// SIMATIC STEP 7 (V5.x) project AmPackRackWIP
// CPU: CPU 315F-2 PN/DP
// CPU: CPU 315F-2 PN/DP
// CPU: CPU 315F-2 PN/DP
// CPU: CPU 315F-2 PN/DP
// CPU: CPU 315F-2 PN/DP
// CPU: CPU 315F-2 PN/DP
// CPU: CPU 315F-2 PN/DP
// station: P_ADR_BUS
// station: _S7H_BUSSYSTEM_CT
// station: SIMATIC Central
// station: Hardware
// station: P_ADR_BUS
// station: SIMATIC Trolley 1
// station: Hardware
// station: P_ADR_BUS
// station: SIMATIC Carrrier 1
// station: Hardware
// station: P_ADR_BUS
// station: SIMATIC Carrrier 2
// station: Hardware
// station: P_ADR_BUS
// station: SIMATIC Trolley 2
// station: Hardware
// station: P_ADR_BUS
// station: SIMATIC Trolley 3
// station: Hardware
// station: P_ADR_BUS
// station: Konfiguration
// station: Hardware
// station: SIMATIC Pegasus
// station: P_ADR_BUS
// station: _S7H_BUSSYSTEM_CT
// program: S7-TR03
// program: S7-MAIN
// program: S7-TR01
// program: S7-CAR01
// program: S7-CAR02
// program: S7-TR02
// program: S7-Programm(7)

SYMBOL_TABLE
"IDB_SafeMain"	DB 1	FB 1
"DB_BRI"	DB 5	DB 5
"DB_ComGateway"	DB 10	DB 10
"IDB_FB2_BRI"	DB 11	FB 2
"DB_OrderBuffer"	DB 15	DB 15
"DB_TargetData"	DB 19	DB 19
"IDB_MasterInterface"	DB 33	FB 13
"IDB_WREC_BR"	DB 50	SFB 53
"INOUT"	DB 80	DB 80
"Moves"	DB 101	DB 101
"InstanzDB PNIODiag"	DB 126	FB 126
"InstanzDB STATDiag"	DB 127	DB 127
"DB_Steps"	DB 132	DB 132
"COMM_CAR01"	DB 150	DB 150
"BRI_Positions"	DB 200	DB 200
"ProfiNET"	DB 400	DB 400
"Error_Safety"	DB 410	DB 410
"IDB_ESTOP1"	DB 415	FB 215
"F_GLOBDB"	DB 545	DB 545	// F_: F_Global_Data Block
"F00020_4FDI_4FDO_iPar"	DB 546	FB 272
"F00025_4FDI_iPar"	DB 547	FB 272
"DB_GLOBAL"	DB 550	DB 550
"F_IO"	DB 690	DB 690
"F_GBL_RECV"	DB 750	DB 750
"IDB_F_RCV"	DB 751	FB 226
"F_GBL_SEND"	DB 752	DB 752
"IDB_F_SND"	DB 753	FB 225
"IDB_WagoiPar_BRI"	DB 920	FB 37
"DB_iPar_Diag"	DB 930	FB 101
"iPar_Data_Bridge"	DB 1920	DB 1920
"SafeMain"	FB 1	FB 1
"MovidriveB_Control"	FB 2	FB 2
"MasterInterface"	FB 13	FB 13
"CheckEncoder"	FB 21	FB 21
"WAGO_iPar_UDL_4_Mod"	FB 37	FB 37	// WAGO up- / download iParameter PROFIsafe Modules
"TSEND"	FB 63	FB 63	// Send Data
"TRCV"	FB 64	FB 64	// Receive Data
"TCON"	FB 65	FB 65	// Connect
"TDISCON"	FB 66	FB 66	// Disconnect
"Safety_Position"	FB 70	FB 70	// Sichere Positionsüberwachung
"Safety_Direction"	FB 72	FB 72	// Sichere Richtungserfassung
"Safety_Speed"	FB 73	FB 73	// Sichere Geschwindigkeit
"Safety_SpeedCheck"	FB 74	FB 74
"Wago_Bridge"	FB 80	FB 80
"F_Input_MAP"	FB 91	FB 91
"ESTOP"	FB 92	FB 92
"GetPos"	FB 93	FB 93
"DiagPROFIsafe_V2_iPar"	FB 101	FB 101	// read diagnosis data of PROFIsafe modules V2 iPar
"PNIODiag"	FB 126	FB 126	// Profibus/DP und Profinet/IO-Diagnose
"STATDiag"	FB 127	FB 127	// Zweitbaustein (PNIODiag)
"F_TON"	FB 185	FB 185	// F_: Timer Switch On Delay
"F_TOF"	FB 186	FB 186	// F_: Timer Switch Off Delay
"F_ESTOP1"	FB 215	FB 215	// F_: Emergency Stop / Stop Category 1
"F_ACK_GL"	FB 219	FB 219	// F_: Global Acknowledgement of all F-I/O of a RTG
"F_SENDS7"	FB 225	FB 225	// F_: Send S7 Connection
"F_RCVS7"	FB 226	FB 226	// F_: Receive S7 Connection
"F_IO_CGP"	FB 272	FB 272	// F_: Driver Block In-Output with Channel Granular Passivation
"F_CTRL_1"	FB 273	FB 273
"F_CTRL_2"	FB 274	FB 274	// F_: Test Block an Programm Run Control
"F_DIAG_N"	FB 275	FB 275	// F_: Diagnosticbuffer Message with non CPU-Stop
"FITON"	FB 276	FB 276	// FI: Timer Switch On Delay
"FITOF"	FB 277	FB 277	// FI: Timer Switch Off Delay
"FIACK_GL"	FB 278	FB 278	// FI: Global Acknowledgement of all F-I/O of a RTG
"F-CALL"	FC 1	FC 1
"Init"	FC 2	FC 2
"AG_SEND"	FC 5	FC 5	// AG SEND
"AG_RECV"	FC 6	FC 6	// AG RECEIVE
"DT_TOD"	FC 8	FC 8	// DT to TOD
"OpHours"	FC 9	FC 9
"EQ_STRNG"	FC 10	FC 10	// Equal String
"AbsEncoder"	FC 11	FC 11
"DT to DATE"	FC 15	FC 15	// DT to DATE
"Inputs"	FC 30	FC 30
"Outputs"	FC 31	FC 31
"Errors"	FC 40	FC 40
"Errors Reset"	FC 41	FC 41
"Errors_001-016_GEN1"	FC 42	FC 42
"Errors_017-032_GEN2"	FC 43	FC 43
"Errors_033-048_NET"	FC 44	FC 44
"EOff_MachineOff"	FC 48	FC 48
"OP_Mode"	FC 49	FC 49
"Send_Buffer"	FC 52	FC 52
"MSG_161-176"	FC 55	FC 55
"MSG_177_192"	FC 56	FC 56
"CheckWindowDi"	FC 100	FC 100
"Communication"	FC 103	FC 103
"STEPS_Control"	FC 110	FC 110
"STEPS_OrderData"	FC 111	FC 111
"STEPS_EMPTY"	FC 113	FC 113
"Axis_BRIDGE"	FC 200	FC 200
"Axis_BRIDGE_Release"	FC 201	FC 201
"Axis_BRIDGE_Control"	FC 202	FC 202
"Axis_BRIDGE_Speed"	FC 203	FC 203
"Axis_BRIDGE_Scan"	FC 204	FC 204
"Axis_BRIDGE_ScanMan"	FC 205	FC 205
"Axis_BRIDGE_Flt_049-064"	FC 209	FC 209
"iPar_ServerCall"	FC 900	FC 900
"BRIGetPosVal_New"	FC 1071	FC 1071
"I_BRI_EStop"	I 20.0	BOOL	// Emergency-Stop tripped
"I_BRI_FB_FastStop"	I 20.1	BOOL	// Feedback safestop bridge
"I_BRI_FB_EStop_CH1"	I 20.2	BOOL	// Feedback E-Stop  CH1
"I_BRI_FB_EStop_CH2"	I 20.3	BOOL	// Feedback E-Stop CH2
"I_BRI_TROinParkp_CH1"	I 25.0	BOOL	// Trolley in Park position CH1
"I_BRI_TROinParkp_CH2"	I 25.1	BOOL	// Trolley in Park position CH1
"I_BRI_Brake_OK"	I 25.2	BOOL	// Temperature Brake resistors OK
"E      25.3"	I 25.3	BOOL	// spare
"I_BRI_BTN_Preset"	I 65.0	BOOL	// preset button
"I_BRI_Fuse24VOK"	I 65.1	BOOL	// fuse 24V DC OK
"I_BRI_temp_cabinet_high"	I 65.2	BOOL	// high temperature cabinet
"I_BRI_Power_BrakesOK"	I 65.3	BOOL	// Power supply brakes OK
"I_BRI_Power_480_OK"	I 65.4	BOOL	// Power supply 480V OK
"I_BRI_Power_Fan"	I 65.5	BOOL	// Power supply fan OK
"I_BRI_BTN_Reset"	I 65.6	BOOL	// reset button
"I_BRI_Fan_active"	I 65.7	BOOL	// Fan is active
"I_BRI_LimitSw_Plus"	I 66.0	BOOL	// Bridge : Limit-Switch Plus
"I_BRI_LimitSw_Minus"	I 66.1	BOOL	// Bridge : Limit-Switch Minus
"I_BRI_FS_PlusNO"	I 66.2	BOOL	// Bridge : forced speed reduction Plus NO
"I_BRI_FS_PlusNC"	I 66.3	BOOL	// Bridge : forced speed reduction Plus NC
"I_BRI_FS_MinusNO"	I 66.4	BOOL	// Bridge : forced speed reduction Minus NO
"I_BRI_FS_MinusNC"	I 66.5	BOOL	// Bridge : forced speed reduction Minus NC
"E      66.6"	I 66.6	BOOL	// spare
"E      66.7"	I 66.7	BOOL	// spare
"E      67.0"	I 67.0	BOOL	// temp. RC plus
"E      67.1"	I 67.1	BOOL	// temp. RC minus
"E      67.2"	I 67.2	BOOL	// temp. RC fast plus
"E      67.3"	I 67.3	BOOL	// temp. RC fast minus
"E      67.4"	I 67.4	BOOL	// spare
"E      67.5"	I 67.5	BOOL	// spare
"E      67.6"	I 67.6	BOOL	// spare
"E      67.7"	I 67.7	BOOL	// spare
"I_BR_ABS_Encoder"	ID 220	DWORD
"OFF"	M 0.0	BOOL	// immer aus
"ON"	M 0.1	BOOL	// immer ein
"FIRST_RUN"	M 0.7	BOOL
"ModeService"	M 1.0	BOOL
"ModeManual"	M 1.1	BOOL
"ModeAuto"	M 1.2	BOOL
"ModeBypass"	M 1.3	BOOL
"ModeServiceOrManual"	M 1.4	BOOL
"StartAuto"	M 1.5	BOOL
"ModeAutoOrManual"	M 1.6	BOOL
"LifeBitMasterOK"	M 1.7	BOOL
"Eoff"	M 2.0	BOOL
"DivEoff"	M 2.1	BOOL
"Error"	M 2.2	BOOL
"Safty_Vorne"	M 2.4	BOOL
"Safty_Hinten"	M 2.5	BOOL
"Safty_Area"	M 2.6	BOOL
"EmOffRelais_delayed"	M 3.0	BOOL
"Clock0_1"	M 10.0	BOOL	// CPU-Takt 0,1s
"Clock0_2"	M 10.1	BOOL	// CPU-Takt 0,2s
"Clock0_4"	M 10.2	BOOL	// CPU-Takt 0,4s
"Clock0_5"	M 10.3	BOOL	// CPU-Takt 0,5s
"Clock0_8"	M 10.4	BOOL	// CPU-Takt 0,8s
"Clock1_0"	M 10.5	BOOL	// CPU-Takt 1,0s
"Clock1_6"	M 10.6	BOOL	// CPU-Takt 1,6s
"Clock2_0"	M 10.7	BOOL	// CPU-Takt 2,0s
"Tick0_1"	M 11.0	BOOL	// Impuls 0,1s
"Tick0_2"	M 11.1	BOOL	// Impuls 0,2s
"Tick0_4"	M 11.2	BOOL	// Impuls 0,4s
"Tick0_5"	M 11.3	BOOL	// Impuls 0,6s
"Tick0_8"	M 11.4	BOOL	// Impuls 0,8s
"Tick1_0"	M 11.5	BOOL	// Impuls 1,0s
"Tick1_6"	M 11.6	BOOL	// Impuls 1,6s
"Tick2_0"	M 11.7	BOOL	// Impuls 2,0s
"SysPulse_0_1"	M 12.0	BOOL
"SysPulse_0_2"	M 12.1	BOOL
"SysPulse_0_4"	M 12.2	BOOL
"SysPulse_0_5"	M 12.3	BOOL
"SysPulse_0_8"	M 12.4	BOOL
"SysPulse_1_0"	M 12.5	BOOL
"SysPulse_1_6"	M 12.6	BOOL
"SysPulse_2_0"	M 12.7	BOOL
"Next_Step"	M 44.0	BOOL
"SingleStep_ON"	M 44.1	BOOL
"One_Single_Step"	M 44.2	BOOL
"BRI_iPar_Check"	M 920.0	BOOL
"BRI_iPar_UpLoad"	M 920.1	BOOL
"BRI_iPar_DownL"	M 920.2	BOOL
"BRI_iPar_ReqDiag"	M 920.5	BOOL
"pFL_BR_StartWago"	M 925.1	BOOL
"pFL_BR_EndWago"	M 925.2	BOOL
"pFl_ResetErrors"	M 1201.2	BOOL
"pFl_13"	M 1201.3	BOOL
"pFl_14"	M 1201.4	BOOL
"pFl_CNT_StartOrder"	M 1202.0	BOOL
"pFl_CNT_EndOrder"	M 1202.1	BOOL
"pFl_SingleNext"	M 1510.0	BOOL
"Bruno_B"	M 2013.0	BOOL	// Programmpunkt muss noch bearbeitet werden
"bTemp0"	MB 20	BYTE
"diTemp00"	MD 20	DWORD
"ENC_Process"	MD 84	DWORD
"CPY_DATETIME_1"	MD 830	DWORD
"CPY_DATETIME_2"	MD 834	DWORD
"BRI_Pos_Motor"	MD 1000	DWORD
"BRI_Pos_Encoder"	MD 1004	DWORD
"CntMsg"	MW 120	INT
"BRI_Motor_HIGH"	MW 1000	INT
"BRI_Motor_LOW"	MW 1002	INT
"BRI_Encoder_HIGH"	MW 1004	INT
"BRI_Encoder_LOW"	MW 1006	INT
"Bruno_W1"	MW 2014	WORD	// Schmierwort
"Bruno_W2"	MW 2016	WORD	// Schmierwort
"Cycle"	OB 1	OB 1
"CYC_INT5"	OB 35	OB 35	// Cyclic Interrupt 5
"I/O_FLT1"	OB 82	OB 82	// I/O Point Fault 1
"I/O_FLT2"	OB 83	OB 83	// I/O Point Fault 2
"OBNL_FLT"	OB 85	OB 85	// OB Not Loaded Fault
"RACK_FLT"	OB 86	OB 86	// Loss of Rack Fault
"COMM_FLT"	OB 87	OB 87	// Communication Fault
"STARTUP"	OB 100	OB 100
"PROG_ERR"	OB 121	OB 121	// Programming Error
"MOD_ERR"	OB 122	OB 122	// Module Access Error
"A      20.0"	Q 20.0	BOOL	// spare
"O_BRI_SafeStop"	Q 20.1	BOOL	// Fast-Stop bridge
"O_BRI_SafeEStop_CH1"	Q 20.2	BOOL	// E-Stop bridge CH1
"O_BRI_SafeEStop_CH2"	Q 20.3	BOOL	// E-Stop bridge CH2
"O_BRI_LP_Preset"	Q 65.0	BOOL	// lamp preset button
"O_BRI_Reset_24V"	Q 65.1	BOOL	// fuse 24VDC reset
"O_BRI_Reset_EStop"	Q 65.2	BOOL	// EStop reset
"O_BRI_LP_Reset"	Q 65.3	BOOL	// lamp reset button
"O_BRI_Horn"	Q 65.4	BOOL	// startup warning
"O_BRI_State_0"	Q 65.5	BOOL	// lamp state 0
"O_BRI_State_1"	Q 65.6	BOOL	// lamp state 1
"O_BRI_State_2"	Q 65.7	BOOL	// lamp state 2
"TON"	SFB 4	SFB 4	// Generate an On Delay
"USEND"	SFB 8	SFB 8	// Uncoordinated Sending of Data
"URCV"	SFB 9	SFB 9	// Uncoordinated Receiving of Data
"RDREC"	SFB 52	SFB 52	// Read a Process Data Record
"WRREC"	SFB 53	SFB 53	// Write a Process Data Record
"RALRM"	SFB 54	SFB 54	// Receive Alarm Data
"GADR_LGC"	SFC 5	SFC 5	// Query Logical Address of a Channel
"RD_SINFO"	SFC 6	SFC 6	// Read OB Start Information
"D_ACT_DP"	SFC 12	SFC 12	// Deactivating and Activating DP Slaves
"DPNRM_DG"	SFC 13	SFC 13	// Read Diagnostic Data of a DP Slave
"DPRD_DAT"	SFC 14	SFC 14	// Read Consistent Data of a Standard DP Slave
"DPWR_DAT"	SFC 15	SFC 15	// Write Consistent Data to a Standard DP Slave
"BLKMOV"	SFC 20	SFC 20	// Copy Variables
"FILL"	SFC 21	SFC 21	// Initialize a Memory Area
"CREAT_DB"	SFC 22	SFC 22	// Create Data Block
"DEL_DB"	SFC 23	SFC 23	// Delete Data Block
"TEST_DB"	SFC 24	SFC 24	// Test Data Block
"DIS_AIRT"	SFC 41	SFC 41	// Delay the Higher Priority Interrupts and Asynchronous Errors
"EN_AIRT"	SFC 42	SFC 42	// Enable Higher Priority Interrupts and Asynchronous Errors
"STP"	SFC 46	SFC 46	// Change the CPU to STOP
"LGC_GADR"	SFC 49	SFC 49	// Query the Module Slot Belonging to a Logical Address
"RDSYSST"	SFC 51	SFC 51	// Read a System Status List or Partial List
"WR_REC"	SFC 58	SFC 58	// Write Data Record
"RD_REC"	SFC 59	SFC 59	// Read a Data Record
"TIME_TCK"	SFC 64	SFC 64	// Read the System Time
"GEO_LOG"	SFC 70	SFC 70	// Determine Logical Address
"LOG_GEO"	SFC 71	SFC 71	// Determine Geographical Address
"tPlcOn"	T 1	TIMER
"tAknowl"	T 2	TIMER
"t_DelEmOffRelais_1"	T 10	TIMER
"t_DelEmOffRelais_2"	T 11	TIMER
"t_BRIDelFastStop"	T 14	TIMER
"t_BRIDelayInPos"	T 15	TIMER
"t_BRIChkRuntime"	T 16	TIMER
"S_Ev_Mes_Auto"	T 18	TIMER
"T_BRI_Preset_SEW"	T 30	TIMER
"T_Delay:PN_01"	T 40	TIMER
"T_Delay:PN_02"	T 41	TIMER
"T_Delay:PN_03"	T 42	TIMER
"t_DelayReadyOnline"	T 60	TIMER
"t_STEPS_start_DEL"	T 70	TIMER
"T_Startup_Warning"	T 94	TIMER
"T_Startup_Horn"	T 95	TIMER
"T_Check_BRI_FS_Minus"	T 150	TIMER
"T_Check_BRI_FS_Plus"	T 151	TIMER
"t_Err_012"	T 212	TIMER
"t_Err_015"	T 215	TIMER
"t_BRI_EStop"	T 220	TIMER
"OneMove"	UDT 7	UDT 7
"HookData"	UDT 100	UDT 100
"HookDataSheet"	UDT 102	UDT 102
"PosCarrier"	VAT 1	
"TestAuto"	VAT 2	
"TestAGV"	VAT 3	
END_SYMBOL_TABLE

TYPE "OneMove"	// UDT 7
VERSION : 0.1
  STRUCT
   MsgCounter : INT ;
   Action : INT ;
   Value_01 : INT ;
   Value_02 : INT ;
   Value_03 : INT ;
   Value_04 : INT ;
   Value_05 : INT ;
   Value_06 : INT ;
   Value_07 : INT ;
   Value_08 : INT ;
   Value_09 : INT ;
   Value_10 : INT ;
   CRC : INT ;
  END_STRUCT ;	
END_TYPE

TYPE "HookData"	// UDT 100
VERSION : 0.1
  STRUCT
   HookType : INT ;
   TotLengthMin : INT ;
   TotLengthMax : INT ;
   FaceLengthMax : INT ;
   CircumMax : INT ;
   TelPos : DINT ;
   Reserve1 : INT ;
  END_STRUCT ;	
END_TYPE

TYPE "HookDataSheet"	// UDT 102
VERSION : 0.1
  STRUCT
   HookOver : DINT ;
   HookUnderOffset : DINT ;
   TelPos_1 : UDT 100;
   TelPos_2 : UDT 100;
   TelPos_3 : UDT 100;
  END_STRUCT ;	
END_TYPE

FUNCTION_BLOCK "SafeMain"	// FB 1
TITLE = Safe Main
AUTHOR : Koenig
VERSION : 0.1
VAR
  ON : BOOL ;
  M_Reset : BOOL ;
  M_Automatic : BOOL ;
  HardwareOK : BOOL ;
  StateOK : BOOL ;
  ESTOP : BOOL ;
  ESTOP_DEL : BOOL ;
  Release_Bridge : BOOL ;
  BRI_STO : BOOL ;
  BRI_Valid : BOOL ;
  BRI_Work : BOOL ;
  Release_STO : BOOL ;
  nFL_STO : BOOL ;
  BRI_SafeAxis : INT ;
  BRI_Pos : INT ;
  ResetGBL : BOOL ;
  RequestGBL : BOOL ;
  SubsGBL : BOOL ;
  WagoBridge : FB 80;
  F_IO : FB 91;
  E_Stop : FB 92;
  ACK : FB 219;
  TOF_STO : FB 186;
  BRI_SafePos : FB 70;
  T_Reset_GBL : FB 185;
  GetPosCarrier : FB 93;
  ErrorArea : BOOL ;
END_VAR
BEGIN
// body was compiled from another editor; compiled code not shown
END_FUNCTION_BLOCK

FUNCTION_BLOCK "MovidriveB_Control"	// FB 2
TITLE = MovidriveB_Control
//main control for the SEW controller
//KNOW_HOW_PROTECT 
//
AUTHOR : Koenig
VERSION : 0.1
VAR_INPUT
  StateWord : INT ;
  FastStop : BOOL ;
  Reset : BOOL ;
  Start : BOOL ;
  InchMinus : BOOL ;
  InchPlus : BOOL ;
  ModeService : BOOL ;
  ModeAuto : BOOL ;
  ModeRef : BOOL ;
  Bypass : BOOL ;
  PlcOn : BOOL ;
  Pulse_1_0 : BOOL ;
  Tick_0_1 : BOOL ;
  ActualPosition : DINT ;
  TargetPosition : DINT ;
  TargetPositionNo : INT ;
  LimitPlus : DINT ;
  LimitMinus : DINT ;
  InPosWin : DINT ;
END_VAR
VAR_OUTPUT
  CrtWord : INT ;
  Moves : BOOL ;
  Ready : BOOL ;
  RefOk : BOOL ;
  InPos : BOOL ;
  BrakeOpen : BOOL ;
  Error : BOOL ;
  ErrCode : INT ;
  ActPosition : DINT ;
  ActPositionNo : INT ;
  ActTarget : DINT ;
END_VAR
VAR
  INT_iCntRelHalt : INT ;
  INT_iCntInPos : INT ;
  INT_ActualPosition : DINT ;
  INT_ActualPositionNo : INT ;
  INT_pFl_ResetPosition : BOOL ;
  INT_TargetOK : BOOL ;
END_VAR
VAR_TEMP
  INT_xStateCode00 : BOOL ;
  INT_xStateCode01 : BOOL ;
  INT_xStateCode02 : BOOL ;
  INT_xStateCode03 : BOOL ;
  INT_xStateCode04 : BOOL ;
  INT_xStateCode05 : BOOL ;
  INT_xStateCode06 : BOOL ;
  INT_xStateCode07 : BOOL ;
  INT_xState : BOOL ;
  INT_xStateReady : BOOL ;
  INT_xStateRefOk : BOOL ;
  INT_xStateInPos : BOOL ;
  INT_xStateNgrNull : BOOL ;
  INT_xStateErrWarn : BOOL ;
  INT_xStateLimitRight : BOOL ;
  INT_xStateLimitLeft : BOOL ;
  INT_xCrtStart : BOOL ;
  INT_xCrtInchPlus : BOOL ;
  INT_xCrtInchMinus : BOOL ;
  INT_xCrtMode11 : BOOL ;
  INT_xCrtMode12 : BOOL ;
  INT_xCrt13 : BOOL ;
  INT_xCrt14 : BOOL ;
  INT_xCrtBypassLimits : BOOL ;
  INT_xCrtLock : BOOL ;
  INT_xCrtRelFaststop : BOOL ;
  INT_xCrtRelHalt : BOOL ;
  INT_xCrtNotPosCrt : BOOL ;
  INT_xCrtRampsSet2 : BOOL ;
  INT_xCrtParaSet2 : BOOL ;
  INT_xCrtReset : BOOL ;
  INT_xCrt06 : BOOL ;
  INT_xModeMan : BOOL ;
  INT_xModeAuto : BOOL ;
  INT_xModeRef : BOOL ;
  INT_ON : BOOL ;
  INT_w00 : WORD ;
  mValue : DINT ;
  pValue : DINT ;
END_VAR
BEGIN
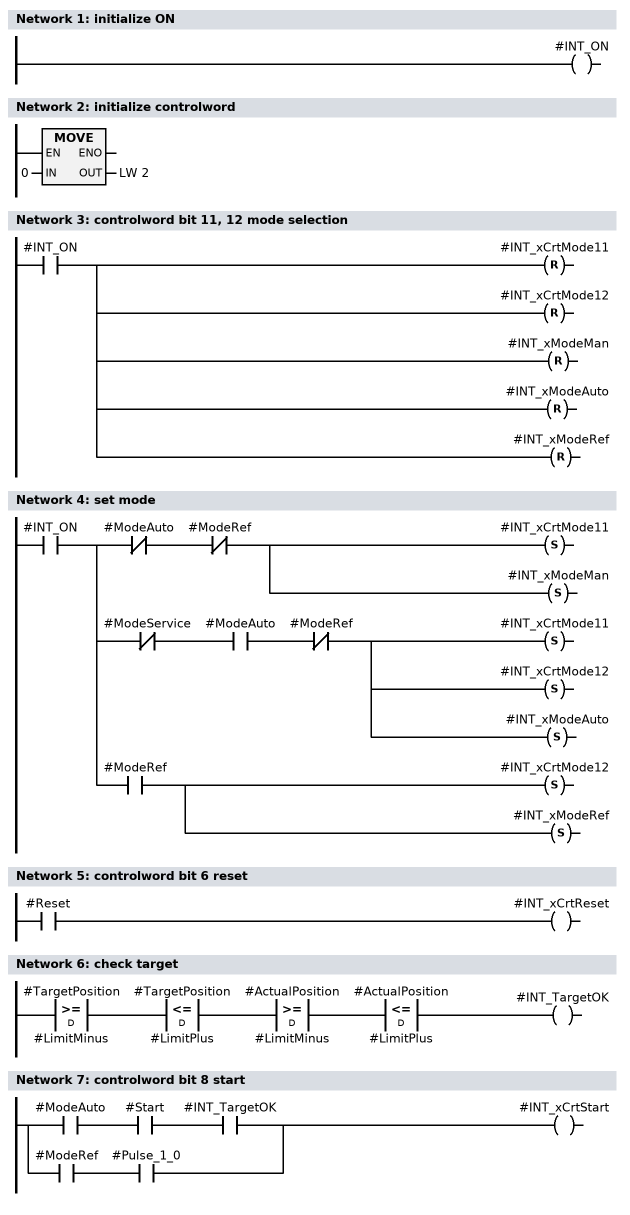
NETWORK
TITLE = initialize ON
//LW0: controler state word
//LW2: controler control word
      SET;
      =     #INT_ON;
NETWORK
TITLE = initialize controlword
      L     0;
      T     LW 2;
      NOP   0;
NETWORK
TITLE = controlword bit 11, 12 mode selection
      A     #INT_ON;
      R     #INT_xCrtMode11;
      R     #INT_xCrtMode12;
      R     #INT_xModeMan;
      R     #INT_xModeAuto;
      R     #INT_xModeRef;
NETWORK
TITLE = set mode
      A     #INT_ON;
      =     L 16.0;
      A     L 16.0;
      AN    #ModeAuto;
      AN    #ModeRef;
      S     #INT_xCrtMode11;
      S     #INT_xModeMan;
      A     L 16.0;
      AN    #ModeService;
      A     #ModeAuto;
      AN    #ModeRef;
      S     #INT_xCrtMode11;
      S     #INT_xCrtMode12;
      S     #INT_xModeAuto;
      A     L 16.0;
      A     #ModeRef;
      S     #INT_xCrtMode12;
      S     #INT_xModeRef;
NETWORK
TITLE = controlword bit 6 reset
      A     #Reset;
      =     #INT_xCrtReset;
NETWORK
TITLE = check target
      A(;
      L     #TargetPosition;
      L     #LimitMinus;
      >=D;
      );
      A(;
      L     #TargetPosition;
      L     #LimitPlus;
      <=D;
      );
      A(;
      L     #ActualPosition;
      L     #LimitMinus;
      >=D;
      );
      A(;
      L     #ActualPosition;
      L     #LimitPlus;
      <=D;
      );
      =     #INT_TargetOK;
NETWORK
TITLE = controlword bit 8 start
      A     #ModeAuto;
      A     #Start;
      A     #INT_TargetOK;
      O;
      A     #ModeRef;
      A     #Pulse_1_0;
      =     #INT_xCrtStart;
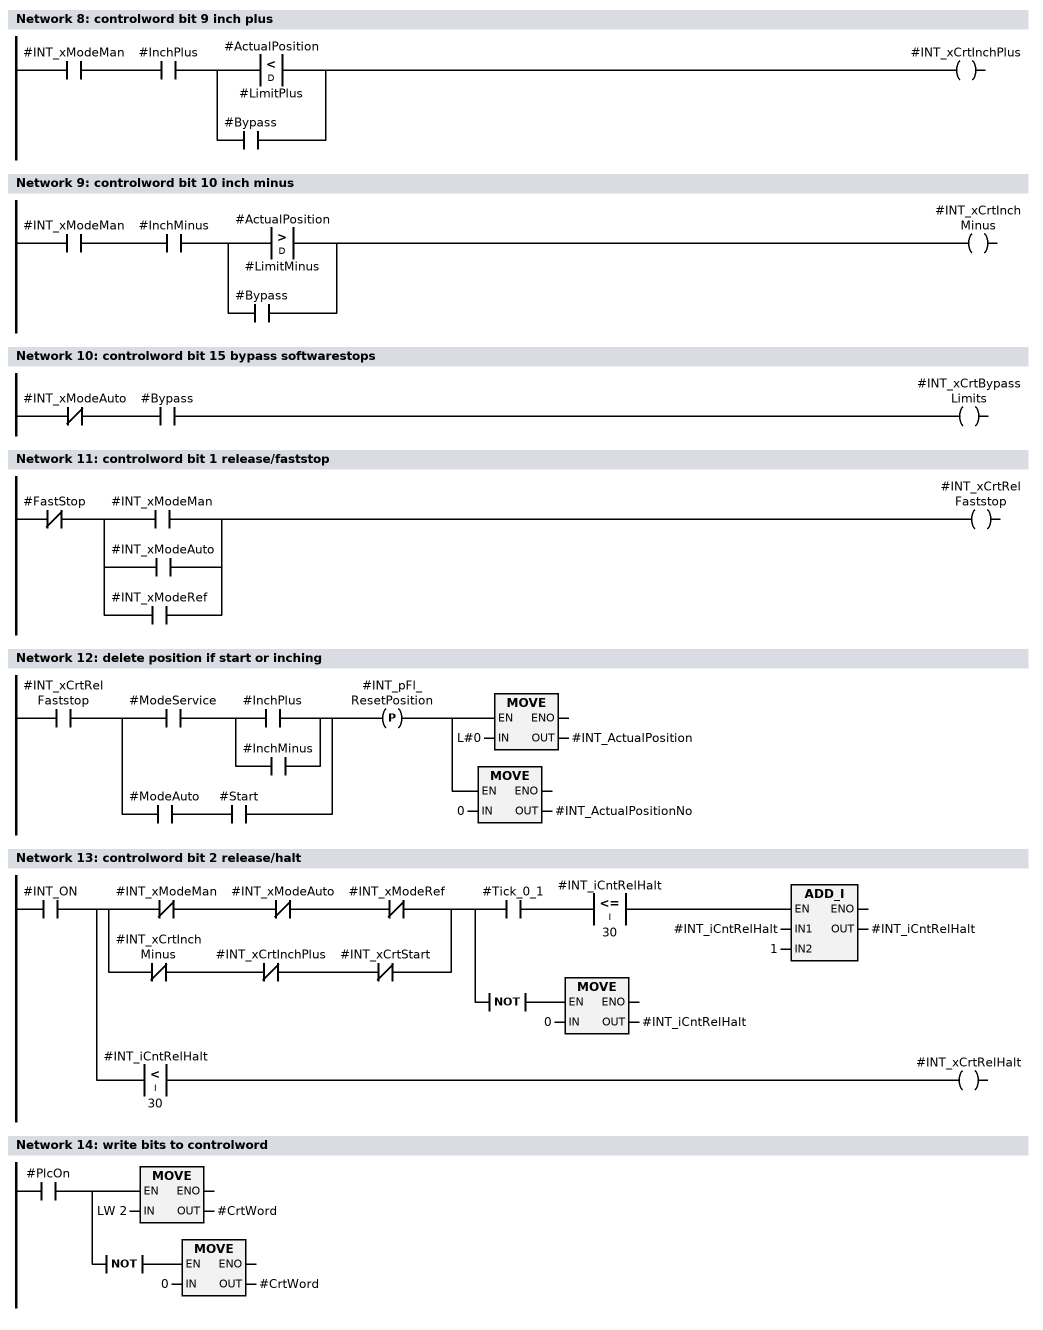
NETWORK
TITLE = controlword bit 9 inch plus
      A     #INT_xModeMan;
      A     #InchPlus;
      A(;
      O(;
      L     #ActualPosition;
      L     #LimitPlus;
      <D;
      );
      O     #Bypass;
      );
      =     #INT_xCrtInchPlus;
NETWORK
TITLE = controlword bit 10 inch minus
      A     #INT_xModeMan;
      A     #InchMinus;
      A(;
      O(;
      L     #ActualPosition;
      L     #LimitMinus;
      >D;
      );
      O     #Bypass;
      );
      =     #INT_xCrtInchMinus;
NETWORK
TITLE = controlword bit 15 bypass softwarestops
      AN    #INT_xModeAuto;
      A     #Bypass;
      =     #INT_xCrtBypassLimits;
NETWORK
TITLE = controlword bit 1 release/faststop
      AN    #FastStop;
      A(;
      O     #INT_xModeMan;
      O     #INT_xModeAuto;
      O     #INT_xModeRef;
      );
      =     #INT_xCrtRelFaststop;
NETWORK
TITLE = delete position if start or inching
      A     #INT_xCrtRelFaststop;
      A(;
      A     #ModeService;
      A(;
      O     #InchPlus;
      O     #InchMinus;
      );
      O;
      A     #ModeAuto;
      A     #Start;
      );
      FP    #INT_pFl_ResetPosition;
      =     L 16.0;
      A     L 16.0;
      JNB   _001;
      L     L#0;
      T     #INT_ActualPosition;
_001: NOP   0;
      A     L 16.0;
      JNB   _002;
      L     0;
      T     #INT_ActualPositionNo;
_002: NOP   0;
NETWORK
TITLE = controlword bit 2 release/halt
      A     #INT_ON;
      =     L 16.0;
      A     L 16.0;
      A(;
      AN    #INT_xModeMan;
      AN    #INT_xModeAuto;
      AN    #INT_xModeRef;
      O;
      AN    #INT_xCrtInchMinus;
      AN    #INT_xCrtInchPlus;
      AN    #INT_xCrtStart;
      );
      =     L 16.1;
      A     L 16.1;
      A     #Tick_0_1;
      A(;
      L     #INT_iCntRelHalt;
      L     30;
      <=I;
      );
      JNB   _003;
      L     #INT_iCntRelHalt;
      L     1;
      +I;
      T     #INT_iCntRelHalt;
_003: NOP   0;
      A     L 16.1;
      NOT;
      JNB   _004;
      L     0;
      T     #INT_iCntRelHalt;
_004: NOP   0;
      A     L 16.0;
      A(;
      L     #INT_iCntRelHalt;
      L     30;
      <I;
      );
      =     #INT_xCrtRelHalt;
NETWORK
TITLE = write bits to controlword
      A     #PlcOn;
      =     L 16.0;
      A     L 16.0;
      JNB   _005;
      L     LW 2;
      T     #CrtWord;
_005: NOP   0;
      A     L 16.0;
      NOT;
      JNB   _006;
      L     0;
      T     #CrtWord;
_006: NOP   0;
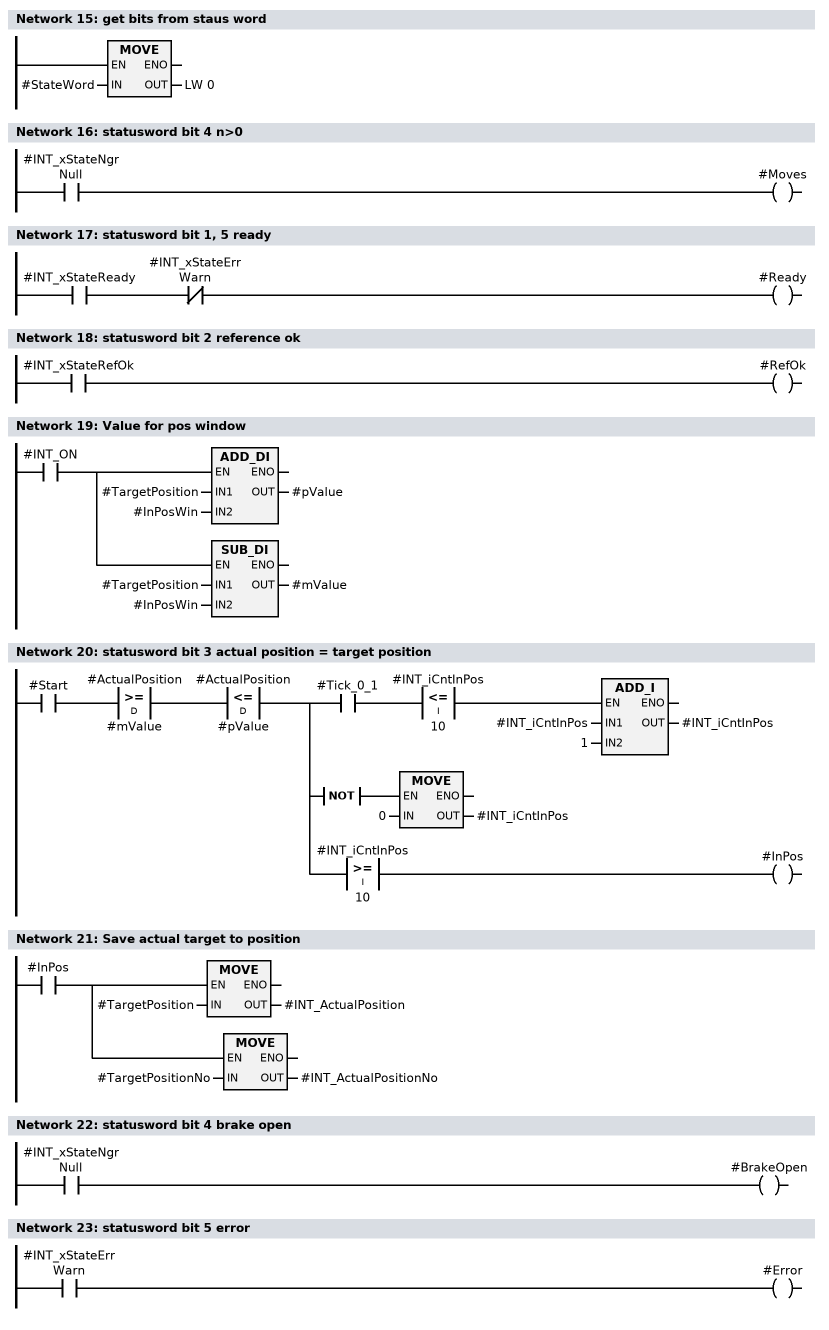
NETWORK
TITLE = get bits from staus word
      L     #StateWord;
      T     LW 0;
      NOP   0;
NETWORK
TITLE = statusword bit 4 n>0
      A     #INT_xStateNgrNull;
      =     #Moves;
NETWORK
TITLE = statusword bit 1, 5 ready
      A     #INT_xStateReady;
      AN    #INT_xStateErrWarn;
      =     #Ready;
NETWORK
TITLE = statusword bit 2 reference ok
      A     #INT_xStateRefOk;
      =     #RefOk;
NETWORK
TITLE = Value for pos window
      A     #INT_ON;
      =     L 16.0;
      A     L 16.0;
      JNB   _007;
      L     #TargetPosition;
      L     #InPosWin;
      +D;
      T     #pValue;
_007: NOP   0;
      A     L 16.0;
      JNB   _008;
      L     #TargetPosition;
      L     #InPosWin;
      -D;
      T     #mValue;
_008: NOP   0;
NETWORK
TITLE = statusword bit 3 actual position = target position
//note: in omron we use the actual position and the target postion equal
//
      A     #Start;
      A(;
      L     #ActualPosition;
      L     #mValue;
      >=D;
      );
      A(;
      L     #ActualPosition;
      L     #pValue;
      <=D;
      );
      =     L 16.0;
      A     L 16.0;
      A     #Tick_0_1;
      A(;
      L     #INT_iCntInPos;
      L     10;
      <=I;
      );
      JNB   _009;
      L     #INT_iCntInPos;
      L     1;
      +I;
      T     #INT_iCntInPos;
_009: NOP   0;
      A     L 16.0;
      NOT;
      JNB   _00a;
      L     0;
      T     #INT_iCntInPos;
_00a: NOP   0;
      A     L 16.0;
      A(;
      L     #INT_iCntInPos;
      L     10;
      >=I;
      );
      =     #InPos;
NETWORK
TITLE = Save actual target to position
      A     #InPos;
      =     L 16.0;
      A     L 16.0;
      JNB   _00b;
      L     #TargetPosition;
      T     #INT_ActualPosition;
_00b: NOP   0;
      A     L 16.0;
      JNB   _00c;
      L     #TargetPositionNo;
      T     #INT_ActualPositionNo;
_00c: NOP   0;
NETWORK
TITLE = statusword bit 4 brake open
      A     #INT_xStateNgrNull;
      =     #BrakeOpen;
NETWORK
TITLE = statusword bit 5 error
      A     #INT_xStateErrWarn;
      =     #Error;
NETWORK
TITLE = status / error code
      A     #INT_ON;
      =     L 16.0;
      A     L 16.0;
      JNB   _00d;
      L     LW 0;
      L     W#16#FF00;
      AW;
      T     LW 0;
_00d: NOP   0;
      A     L 16.0;
      JNB   _00e;
      L     W#16#8;
      L     LW 0;
      SRW;
      T     LW 0;
_00e: NOP   0;
      A     L 16.0;
      JNB   _00f;
      L     LW 0;
      T     #ErrCode;
_00f: NOP   0;
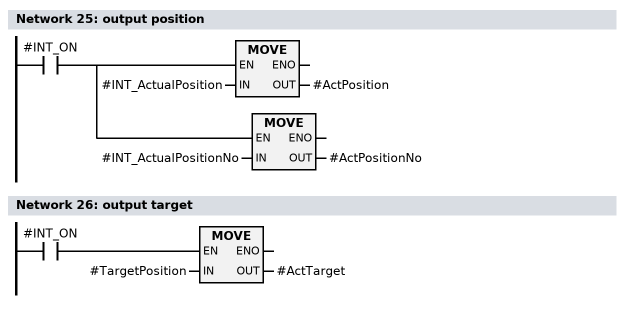
NETWORK
TITLE = output position
      A     #INT_ON;
      =     L 16.0;
      A     L 16.0;
      JNB   _010;
      L     #INT_ActualPosition;
      T     #ActPosition;
_010: NOP   0;
      A     L 16.0;
      JNB   _011;
      L     #INT_ActualPositionNo;
      T     #ActPositionNo;
_011: NOP   0;
NETWORK
TITLE = output target
      A     #INT_ON;
      JNB   _012;
      L     #TargetPosition;
      T     #ActTarget;
_012: NOP   0;
END_FUNCTION_BLOCK

FUNCTION_BLOCK "MasterInterface"	// FB 13
//LW0: control word from master
//LW2: status word to master
VERSION : 0.1
VAR_INPUT
  IN_iCrtWord : INT ;
  IN_iCommCounter : INT ;
  IN_iToggleTime_0_1sec : INT ;
  IN_xFree : BOOL ;
  IN_xOccupied : BOOL ;
  IN_xLiftTop : BOOL ;
  IN_xOnline : BOOL ;
  IN_xReadyOnline : BOOL ;
  IN_xError : BOOL ;
  IN_xMovingSource : BOOL ;
  IN_xMovingTarget : BOOL ;
  IN_x09 : BOOL ;
  IN_xOrderRunning : BOOL ;
  IN_xOrderEnd : BOOL ;
  IN_xOrderPaused : BOOL ;
  IN_x13 : BOOL ;
  IN_xNewTarget : BOOL ;
  IN_x15 : BOOL ;
  IN_SysTick : BOOL ;
END_VAR
VAR_OUTPUT
  OUT_iStateWord : INT ;
  OUT_xLifeBitOk : BOOL ;
  OUT_x01 : BOOL ;
  OUT_xStartBasePos : BOOL ;
  OUT_xStartNewTarget : BOOL ;
  OUT_xAknOrderEnd : BOOL ;
  OUT_xReset : BOOL ;
  OUT_x06 : BOOL ;
  OUT_x07 : BOOL ;
  OUT_x08 : BOOL ;
  OUT_x09 : BOOL ;
  OUT_xStartOrder : BOOL ;
  OUT_xClearOrder : BOOL ;
  OUT_xPauseOrder : BOOL ;
  OUT_x13 : BOOL ;
  OUT_xStartStopPos : BOOL ;
  OUT_xReleaseOnline : BOOL ;
END_VAR
VAR
  INT_b_1 : BOOL ;
  INT_b_2 : BOOL ;
  INT_b_3 : BOOL ;
  INT_iCntLbOn : INT ;
  INT_iCntLbOff : INT ;
  INT_iCntLbOk : INT ;
  INT_iCntStartBasePos : INT ;
  INT_iCntStartNewtarget : INT ;
  INT_iCntStartOrder : INT ;
  INT_iCntStartStopPos : INT ;
  INT_iLastCommCounter : INT ;
  INT_T1 : SFB 4;
  INT_T2 : SFB 4;
END_VAR
VAR_TEMP
  INT_xCrt08 : BOOL ;
  INT_xCrt09 : BOOL ;
  INT_xCrtStartOrder : BOOL ;
  INT_xCrtClearOrder : BOOL ;
  INT_xCrtPauseOrder : BOOL ;
  INT_xCrt13 : BOOL ;
  INT_xCrtStartStopPos : BOOL ;
  INT_xReleaseOnline : BOOL ;
  INT_xCrtLife : BOOL ;
  INT_xCrt01 : BOOL ;
  INT_xCrtStartBasePos : BOOL ;
  INT_xCrtStartNewTarg : BOOL ;
  INT_xCrtAcknOrderEnd : BOOL ;
  INT_xCrtReset : BOOL ;
  INT_xCrt06 : BOOL ;
  INT_xCrt07 : BOOL ;
  INT_xStateMovingTarget : BOOL ;
  INT_xState09 : BOOL ;
  INT_xStateOrderRunning : BOOL ;
  INT_xStateOrderEnd : BOOL ;
  INT_xStateOrderPaused : BOOL ;
  INT_xState13 : BOOL ;
  INT_xStateNewTarget : BOOL ;
  INT_xState15 : BOOL ;
  INT_xStateLife : BOOL ;
  INT_xStateFree : BOOL ;
  INT_xStateOccupied : BOOL ;
  INT_xStateLiftTop : BOOL ;
  INT_xStateOnline : BOOL ;
  INT_xStateReadyOnline : BOOL ;
  INT_xStateError : BOOL ;
  INT_xStateMovingSource : BOOL ;
  ON : BOOL ;
END_VAR
BEGIN
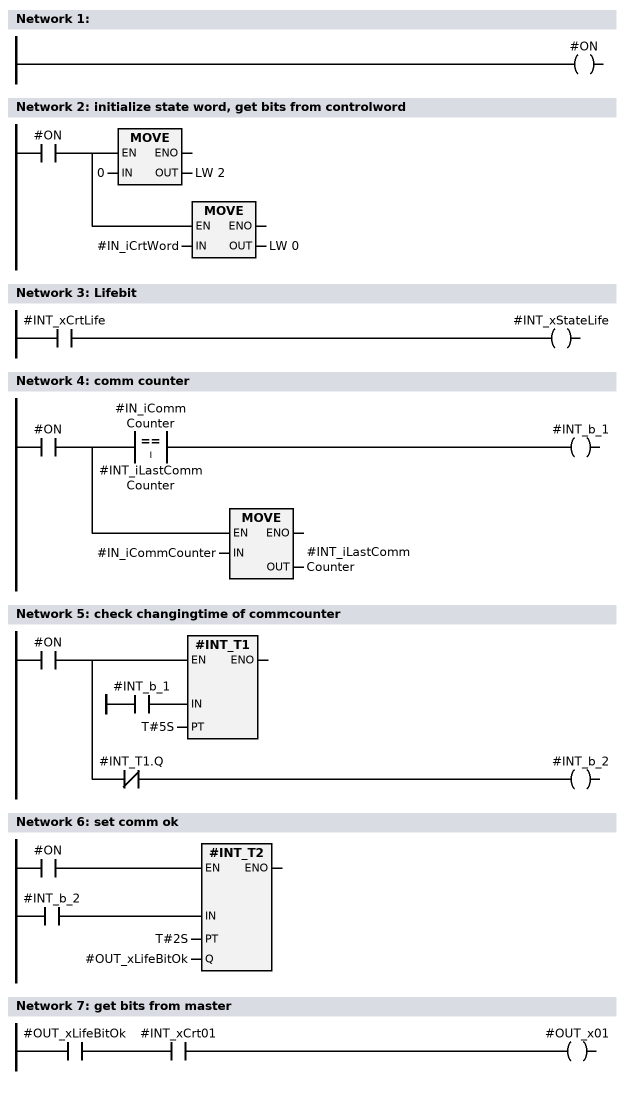
NETWORK
TITLE =
      SET;
      =     #ON;
NETWORK
TITLE = initialize state word, get bits from controlword
      A     #ON;
      =     L 5.0;
      A     L 5.0;
      JNB   _001;
      L     0;
      T     LW 2;
_001: NOP   0;
      A     L 5.0;
      JNB   _002;
      L     #IN_iCrtWord;
      T     LW 0;
_002: NOP   0;
NETWORK
TITLE = Lifebit
      A     #INT_xCrtLife;
      =     #INT_xStateLife;
NETWORK
TITLE = comm counter
      A     #ON;
      =     L 5.0;
      A     L 5.0;
      A(;
      L     #IN_iCommCounter;
      L     #INT_iLastCommCounter;
      ==I;
      );
      =     #INT_b_1;
      A     L 5.0;
      JNB   _003;
      L     #IN_iCommCounter;
      T     #INT_iLastCommCounter;
_003: NOP   0;
NETWORK
TITLE = check changingtime of commcounter
      A     #ON;
      =     L 5.0;
      A     #INT_b_1;
      =     L 5.1;
      BLD   103;
      A     L 5.0;
      JNB   _004;
      CALL  #INT_T1 (
           IN                       := L 5.1,
           PT                       := T#5S);
_004: NOP   0;
      A     L 5.0;
      AN    #INT_T1.Q;
      =     #INT_b_2;
NETWORK
TITLE = set comm ok
      A     #INT_b_2;
      =     L 5.0;
      BLD   103;
      A     #ON;
      JNB   _005;
      CALL  #INT_T2 (
           IN                       := L 5.0,
           PT                       := T#2S,
           Q                        := #OUT_xLifeBitOk);
_005: NOP   0;
NETWORK
TITLE = get bits from master
      A     #OUT_xLifeBitOk;
      A     #INT_xCrt01;
      =     #OUT_x01;
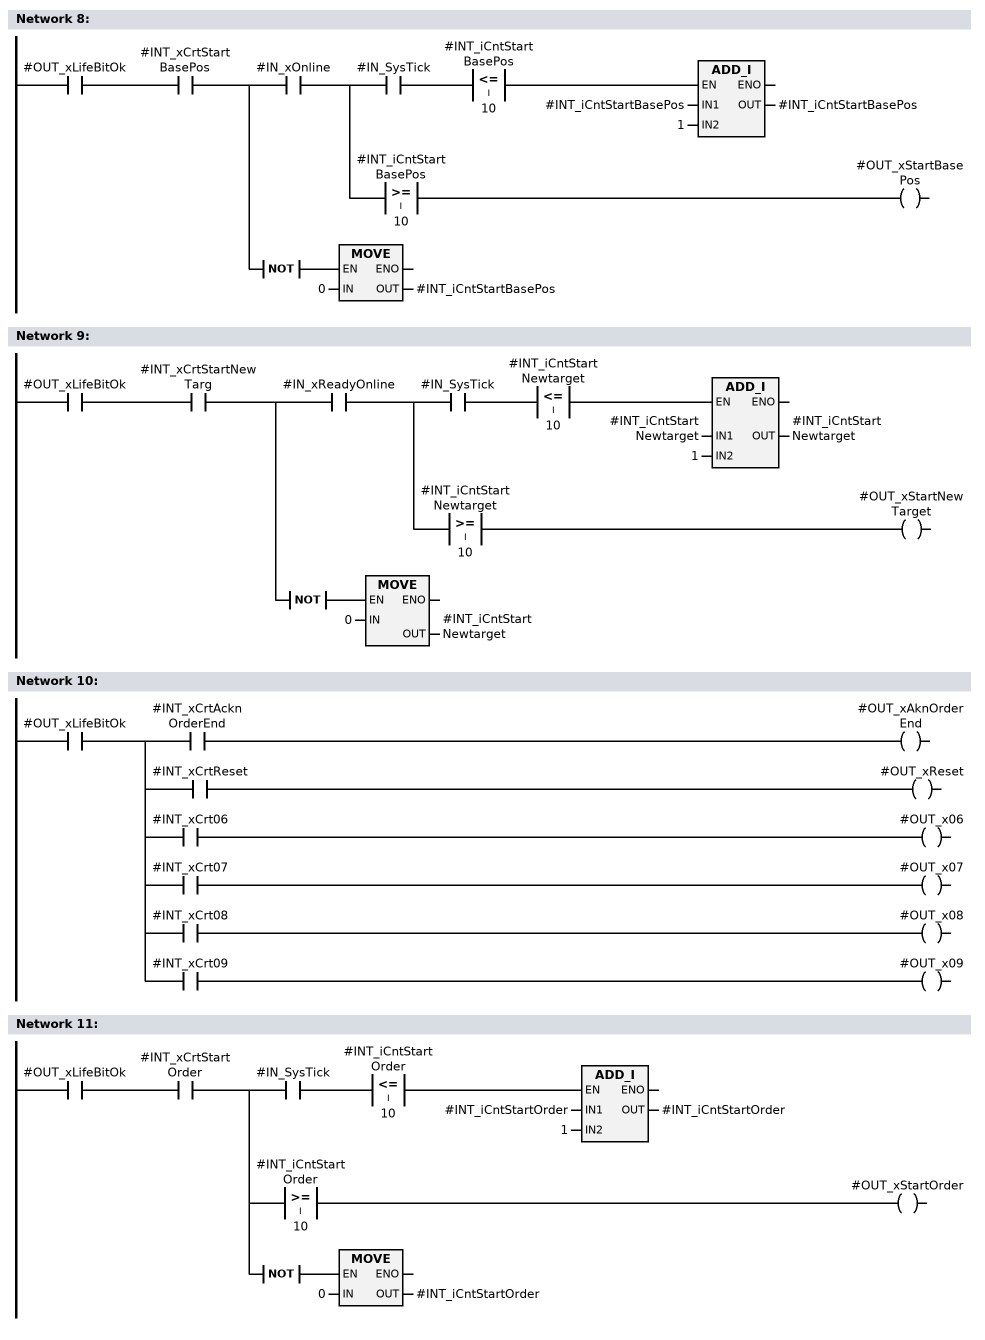
NETWORK
TITLE =
      A     #OUT_xLifeBitOk;
      A     #INT_xCrtStartBasePos;
      =     L 5.0;
      A     L 5.0;
      A     #IN_xOnline;
      =     L 5.1;
      A     L 5.1;
      A     #IN_SysTick;
      A(;
      L     #INT_iCntStartBasePos;
      L     10;
      <=I;
      );
      JNB   _006;
      L     #INT_iCntStartBasePos;
      L     1;
      +I;
      T     #INT_iCntStartBasePos;
_006: NOP   0;
      A     L 5.1;
      A(;
      L     #INT_iCntStartBasePos;
      L     10;
      >=I;
      );
      =     #OUT_xStartBasePos;
      A     L 5.0;
      NOT;
      JNB   _007;
      L     0;
      T     #INT_iCntStartBasePos;
_007: NOP   0;
NETWORK
TITLE =
      A     #OUT_xLifeBitOk;
      A     #INT_xCrtStartNewTarg;
      =     L 5.0;
      A     L 5.0;
      A     #IN_xReadyOnline;
      =     L 5.1;
      A     L 5.1;
      A     #IN_SysTick;
      A(;
      L     #INT_iCntStartNewtarget;
      L     10;
      <=I;
      );
      JNB   _008;
      L     #INT_iCntStartNewtarget;
      L     1;
      +I;
      T     #INT_iCntStartNewtarget;
_008: NOP   0;
      A     L 5.1;
      A(;
      L     #INT_iCntStartNewtarget;
      L     10;
      >=I;
      );
      =     #OUT_xStartNewTarget;
      A     L 5.0;
      NOT;
      JNB   _009;
      L     0;
      T     #INT_iCntStartNewtarget;
_009: NOP   0;
NETWORK
TITLE =
      A     #OUT_xLifeBitOk;
      =     L 5.0;
      A     L 5.0;
      A     #INT_xCrtAcknOrderEnd;
      =     #OUT_xAknOrderEnd;
      A     L 5.0;
      A     #INT_xCrtReset;
      =     #OUT_xReset;
      A     L 5.0;
      A     #INT_xCrt06;
      =     #OUT_x06;
      A     L 5.0;
      A     #INT_xCrt07;
      =     #OUT_x07;
      A     L 5.0;
      A     #INT_xCrt08;
      =     #OUT_x08;
      A     L 5.0;
      A     #INT_xCrt09;
      =     #OUT_x09;
NETWORK
TITLE =
      A     #OUT_xLifeBitOk;
      A     #INT_xCrtStartOrder;
      =     L 5.0;
      A     L 5.0;
      A     #IN_SysTick;
      A(;
      L     #INT_iCntStartOrder;
      L     10;
      <=I;
      );
      JNB   _00a;
      L     #INT_iCntStartOrder;
      L     1;
      +I;
      T     #INT_iCntStartOrder;
_00a: NOP   0;
      A     L 5.0;
      A(;
      L     #INT_iCntStartOrder;
      L     10;
      >=I;
      );
      =     #OUT_xStartOrder;
      A     L 5.0;
      NOT;
      JNB   _00b;
      L     0;
      T     #INT_iCntStartOrder;
_00b: NOP   0;
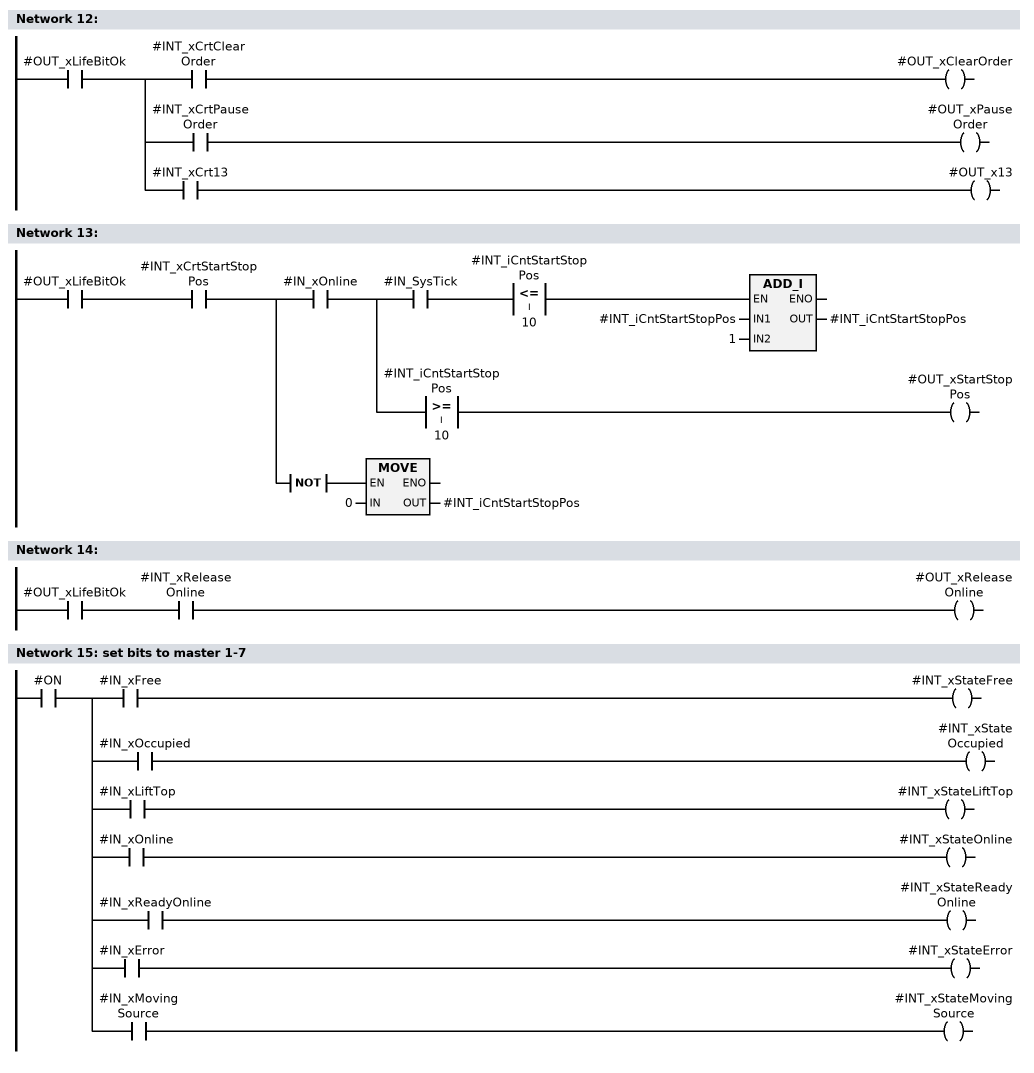
NETWORK
TITLE =
      A     #OUT_xLifeBitOk;
      =     L 5.0;
      A     L 5.0;
      A     #INT_xCrtClearOrder;
      =     #OUT_xClearOrder;
      A     L 5.0;
      A     #INT_xCrtPauseOrder;
      =     #OUT_xPauseOrder;
      A     L 5.0;
      A     #INT_xCrt13;
      =     #OUT_x13;
NETWORK
TITLE =
      A     #OUT_xLifeBitOk;
      A     #INT_xCrtStartStopPos;
      =     L 5.0;
      A     L 5.0;
      A     #IN_xOnline;
      =     L 5.1;
      A     L 5.1;
      A     #IN_SysTick;
      A(;
      L     #INT_iCntStartStopPos;
      L     10;
      <=I;
      );
      JNB   _00c;
      L     #INT_iCntStartStopPos;
      L     1;
      +I;
      T     #INT_iCntStartStopPos;
_00c: NOP   0;
      A     L 5.1;
      A(;
      L     #INT_iCntStartStopPos;
      L     10;
      >=I;
      );
      =     #OUT_xStartStopPos;
      A     L 5.0;
      NOT;
      JNB   _00d;
      L     0;
      T     #INT_iCntStartStopPos;
_00d: NOP   0;
NETWORK
TITLE =
      A     #OUT_xLifeBitOk;
      A     #INT_xReleaseOnline;
      =     #OUT_xReleaseOnline;
NETWORK
TITLE = set bits to master 1-7
      A     #ON;
      =     L 5.0;
      A     L 5.0;
      A     #IN_xFree;
      =     #INT_xStateFree;
      A     L 5.0;
      A     #IN_xOccupied;
      =     #INT_xStateOccupied;
      A     L 5.0;
      A     #IN_xLiftTop;
      =     #INT_xStateLiftTop;
      A     L 5.0;
      A     #IN_xOnline;
      =     #INT_xStateOnline;
      A     L 5.0;
      A     #IN_xReadyOnline;
      =     #INT_xStateReadyOnline;
      A     L 5.0;
      A     #IN_xError;
      =     #INT_xStateError;
      A     L 5.0;
      A     #IN_xMovingSource;
      =     #INT_xStateMovingSource;
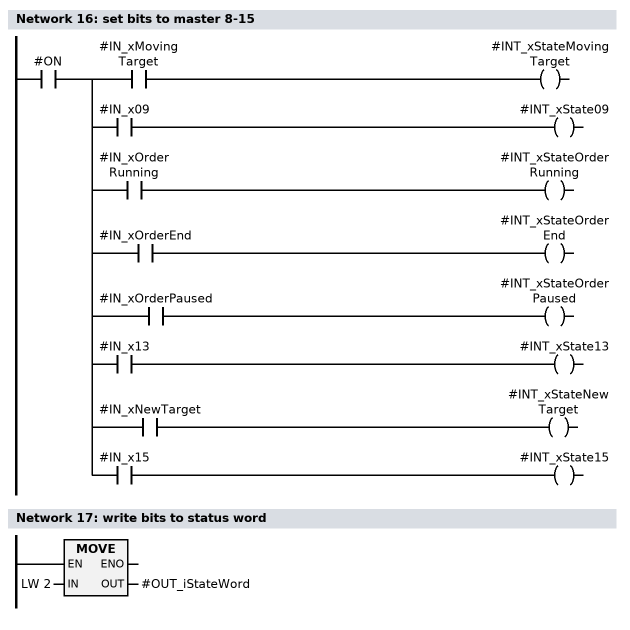
NETWORK
TITLE = set bits to master 8-15
      A     #ON;
      =     L 5.0;
      A     L 5.0;
      A     #IN_xMovingTarget;
      =     #INT_xStateMovingTarget;
      A     L 5.0;
      A     #IN_x09;
      =     #INT_xState09;
      A     L 5.0;
      A     #IN_xOrderRunning;
      =     #INT_xStateOrderRunning;
      A     L 5.0;
      A     #IN_xOrderEnd;
      =     #INT_xStateOrderEnd;
      A     L 5.0;
      A     #IN_xOrderPaused;
      =     #INT_xStateOrderPaused;
      A     L 5.0;
      A     #IN_x13;
      =     #INT_xState13;
      A     L 5.0;
      A     #IN_xNewTarget;
      =     #INT_xStateNewTarget;
      A     L 5.0;
      A     #IN_x15;
      =     #INT_xState15;
NETWORK
TITLE = write bits to status word
      L     LW 2;
      T     #OUT_iStateWord;
      NOP   0;
END_FUNCTION_BLOCK

FUNCTION_BLOCK "CheckEncoder"	// FB 21
TITLE = Check Encoder
VERSION : 0.1
VAR_INPUT
  ActualValue : DINT ;
  TurnMinus : BOOL ;
  TurnPlus : BOOL ;
  Reset : BOOL ;
  Clock_100ms : BOOL ;
  Clock_1s : BOOL ;
  minTurn : DINT ;
  maxTurn : DINT ;
  maxNotTurn : DINT ;
  fadeOut100ms : INT ;
END_VAR
VAR_OUTPUT
  Error : BOOL ;
  ErrorCode : INT ;
END_VAR
VAR
  lastValue : DINT ;
  actDiff : DINT ;
  p_Reset : BOOL ;
  p_Clock : BOOL ;
  p_Clock_1s : BOOL ;
  m_Error : BOOL ;
  timerTurn : INT ;
  timerNotTurn : INT ;
  m_ErrorCode : INT ;
  m_ErrorDiff : DINT ;
  timerCheck : INT ;
END_VAR
VAR_TEMP
  Clock : BOOL ;
  Turn : BOOL ;
  notTurn : BOOL ;
  Clock_1 : BOOL ;
END_VAR
BEGIN
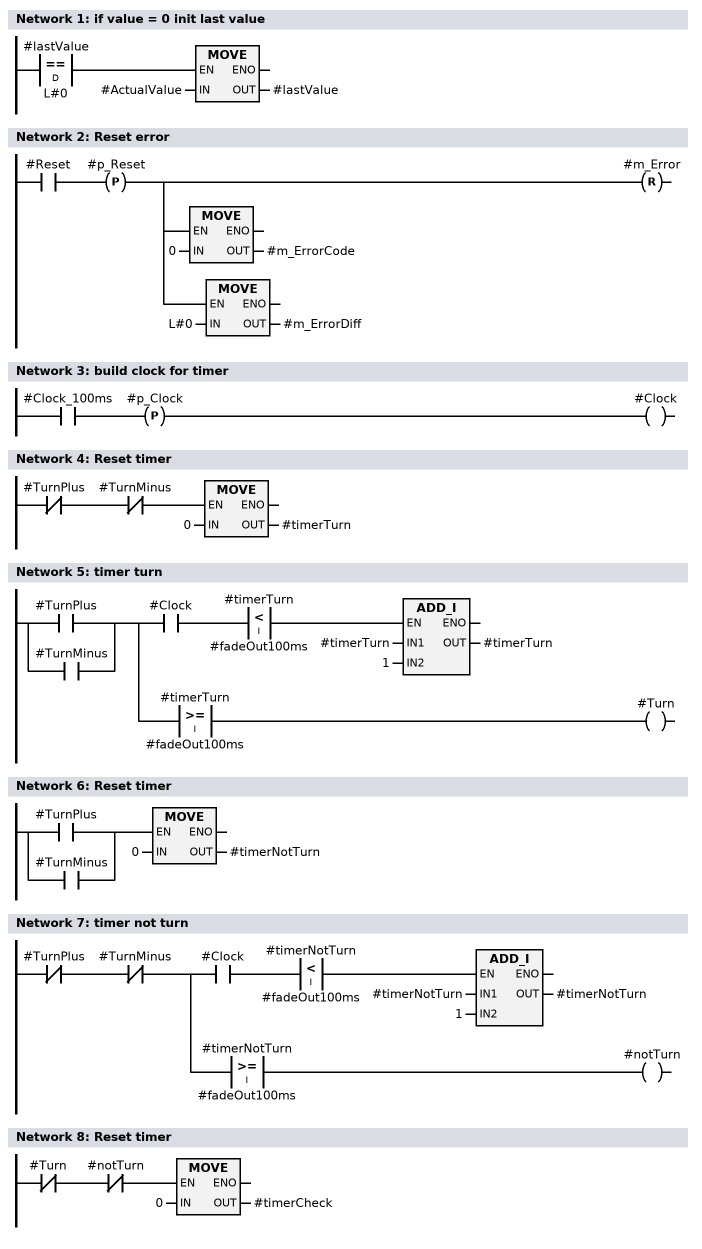
NETWORK
TITLE = if value = 0 init last value
      A(;
      L     #lastValue;
      L     L#0;
      ==D;
      );
      JNB   _001;
      L     #ActualValue;
      T     #lastValue;
_001: NOP   0;
NETWORK
TITLE = Reset error
      A     #Reset;
      FP    #p_Reset;
      =     L 1.0;
      A     L 1.0;
      BLD   102;
      R     #m_Error;
      A     L 1.0;
      JNB   _002;
      L     0;
      T     #m_ErrorCode;
_002: NOP   0;
      A     L 1.0;
      JNB   _003;
      L     L#0;
      T     #m_ErrorDiff;
_003: NOP   0;
NETWORK
TITLE = build clock for timer
      A     #Clock_100ms;
      FP    #p_Clock;
      =     #Clock;
NETWORK
TITLE = Reset timer
      AN    #TurnPlus;
      AN    #TurnMinus;
      JNB   _004;
      L     0;
      T     #timerTurn;
_004: NOP   0;
NETWORK
TITLE = timer turn
      O     #TurnPlus;
      O     #TurnMinus;
      =     L 1.0;
      A     L 1.0;
      A     #Clock;
      A(;
      L     #timerTurn;
      L     #fadeOut100ms;
      <I;
      );
      JNB   _005;
      L     #timerTurn;
      L     1;
      +I;
      T     #timerTurn;
_005: NOP   0;
      A     L 1.0;
      A(;
      L     #timerTurn;
      L     #fadeOut100ms;
      >=I;
      );
      =     #Turn;
NETWORK
TITLE = Reset timer
      A(;
      O     #TurnPlus;
      O     #TurnMinus;
      );
      JNB   _006;
      L     0;
      T     #timerNotTurn;
_006: NOP   0;
NETWORK
TITLE = timer not turn
      AN    #TurnPlus;
      AN    #TurnMinus;
      =     L 1.0;
      A     L 1.0;
      A     #Clock;
      A(;
      L     #timerNotTurn;
      L     #fadeOut100ms;
      <I;
      );
      JNB   _007;
      L     #timerNotTurn;
      L     1;
      +I;
      T     #timerNotTurn;
_007: NOP   0;
      A     L 1.0;
      A(;
      L     #timerNotTurn;
      L     #fadeOut100ms;
      >=I;
      );
      =     #notTurn;
NETWORK
TITLE = Reset timer
      AN    #Turn;
      AN    #notTurn;
      JNB   _008;
      L     0;
      T     #timerCheck;
_008: NOP   0;
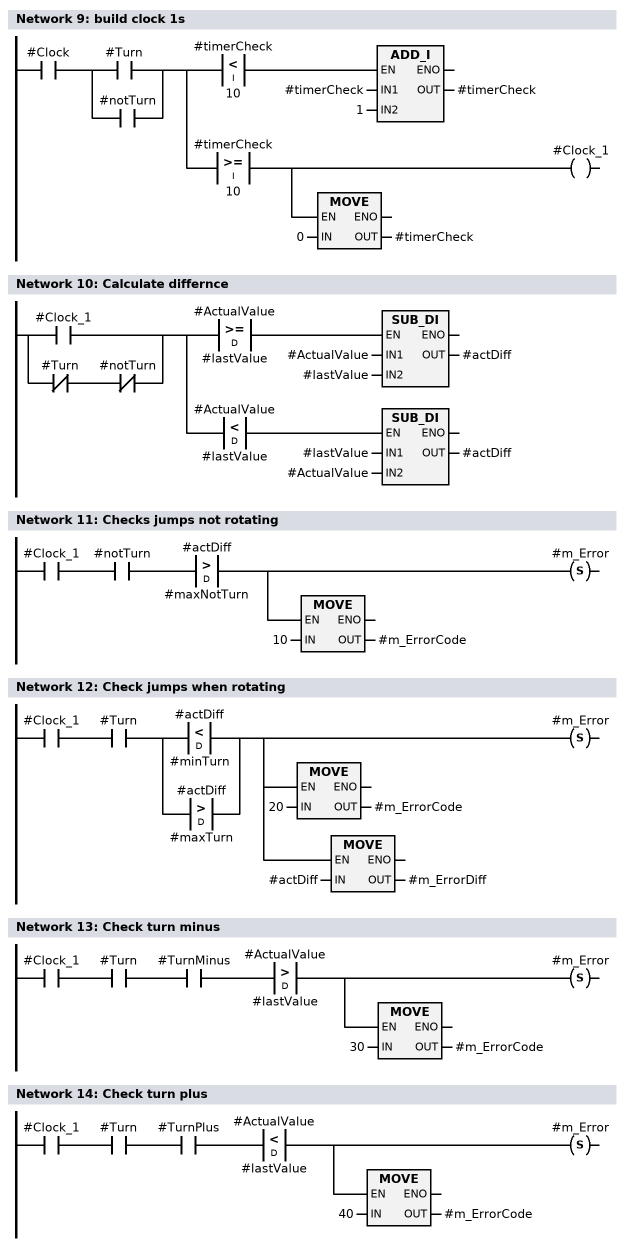
NETWORK
TITLE = build clock 1s
      A     #Clock;
      A(;
      O     #Turn;
      O     #notTurn;
      );
      =     L 1.0;
      A     L 1.0;
      A(;
      L     #timerCheck;
      L     10;
      <I;
      );
      JNB   _009;
      L     #timerCheck;
      L     1;
      +I;
      T     #timerCheck;
_009: NOP   0;
      A     L 1.0;
      A(;
      L     #timerCheck;
      L     10;
      >=I;
      );
      =     L 1.1;
      A     L 1.1;
      BLD   102;
      =     #Clock_1;
      A     L 1.1;
      JNB   _00a;
      L     0;
      T     #timerCheck;
_00a: NOP   0;
NETWORK
TITLE = Calculate differnce
      O     #Clock_1;
      O;
      AN    #Turn;
      AN    #notTurn;
      =     L 1.0;
      A     L 1.0;
      A(;
      L     #ActualValue;
      L     #lastValue;
      >=D;
      );
      JNB   _00b;
      L     #ActualValue;
      L     #lastValue;
      -D;
      T     #actDiff;
_00b: NOP   0;
      A     L 1.0;
      A(;
      L     #ActualValue;
      L     #lastValue;
      <D;
      );
      JNB   _00c;
      L     #lastValue;
      L     #ActualValue;
      -D;
      T     #actDiff;
_00c: NOP   0;
NETWORK
TITLE = Checks jumps not rotating
      A     #Clock_1;
      A     #notTurn;
      A(;
      L     #actDiff;
      L     #maxNotTurn;
      >D;
      );
      =     L 1.0;
      A     L 1.0;
      BLD   102;
      S     #m_Error;
      A     L 1.0;
      JNB   _00d;
      L     10;
      T     #m_ErrorCode;
_00d: NOP   0;
NETWORK
TITLE = Check jumps when rotating
      A     #Clock_1;
      A     #Turn;
      A(;
      O(;
      L     #actDiff;
      L     #minTurn;
      <D;
      );
      O(;
      L     #actDiff;
      L     #maxTurn;
      >D;
      );
      );
      =     L 1.0;
      A     L 1.0;
      BLD   102;
      S     #m_Error;
      A     L 1.0;
      JNB   _00e;
      L     20;
      T     #m_ErrorCode;
_00e: NOP   0;
      A     L 1.0;
      JNB   _00f;
      L     #actDiff;
      T     #m_ErrorDiff;
_00f: NOP   0;
NETWORK
TITLE = Check turn minus
      A     #Clock_1;
      A     #Turn;
      A     #TurnMinus;
      A(;
      L     #ActualValue;
      L     #lastValue;
      >D;
      );
      =     L 1.0;
      A     L 1.0;
      BLD   102;
      S     #m_Error;
      A     L 1.0;
      JNB   _010;
      L     30;
      T     #m_ErrorCode;
_010: NOP   0;
NETWORK
TITLE = Check turn plus
      A     #Clock_1;
      A     #Turn;
      A     #TurnPlus;
      A(;
      L     #ActualValue;
      L     #lastValue;
      <D;
      );
      =     L 1.0;
      A     L 1.0;
      BLD   102;
      S     #m_Error;
      A     L 1.0;
      JNB   _011;
      L     40;
      T     #m_ErrorCode;
_011: NOP   0;
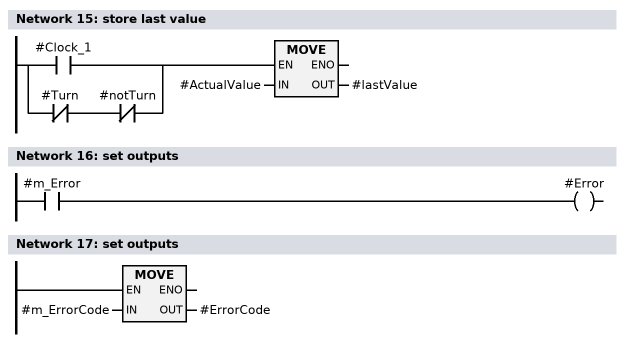
NETWORK
TITLE = store last value
      A(;
      O     #Clock_1;
      O;
      AN    #Turn;
      AN    #notTurn;
      );
      JNB   _012;
      L     #ActualValue;
      T     #lastValue;
_012: NOP   0;
NETWORK
TITLE = set outputs
      A     #m_Error;
      =     #Error;
NETWORK
TITLE = set outputs
      L     #m_ErrorCode;
      T     #ErrorCode;
      NOP   0;
END_FUNCTION_BLOCK

// FB 37: know-how protected block, not included

// FB 63: know-how protected block, not included

// FB 64: know-how protected block, not included

// FB 65: know-how protected block, not included

// FB 66: know-how protected block, not included

FUNCTION_BLOCK "Safety_Position"	// FB 70
TITLE = Check safety positon
AUTHOR : Koenig
VERSION : 0.1
VAR_INPUT
  IN_Encoder_1_LO : INT ;	//Encoder 1 Low Word
  IN_Encoder_1_HI : INT ;	//Encoder 1 High Word
  IN_Encoder_2_LO : INT ;	//Encoder 2 Low Word
  IN_Encoder_2_HI : INT ;	//Encoder 2 High Word
  ReleaseFast : BOOL ;
  DiffSlow : INT ;
  DiffFast : INT ;
  Reset : BOOL ;
  Delay_CHK : TIME  := T#5S;
END_VAR
VAR_OUTPUT
  OUT_Difference_Lo : INT ;
  OUT_Difference_HI : INT ;
  Valid : BOOL ;
  Error_Diff : BOOL ;
END_VAR
VAR
  OFF : BOOL ;
  ON : BOOL ;
  delay : FB 186;
  checkDiff : BOOL ;
  err_Diff : BOOL ;
  delayTime : TIME  := T#1S;
  tmp_Difference_LO : INT ;
  tmp_Difference_HI : INT ;
  tmp_Encoder2_HI : INT ;
  tmp_lowerZero : BOOL ;
  tmp_ovBit_Sub1_LO : BOOL ;
  tmp_ovBit_Sub1_HI : BOOL ;
  tmp_ovBit_Mul1 : BOOL ;
  tmp_OFF : BOOL ;
  tmp_slow : BOOL ;
  chk_slow : BOOL ;
  t_slow : FB 185;
END_VAR
BEGIN
// body was compiled from another editor; compiled code not shown
END_FUNCTION_BLOCK

FUNCTION_BLOCK "Safety_Direction"	// FB 72
TITLE = Check direction
AUTHOR : Koenig
VERSION : 0.1
VAR_INPUT
  ActualPosition : INT ;
END_VAR
VAR_OUTPUT
  DirPlus : BOOL ;
  DirMinus : BOOL ;
  DirStop : BOOL ;
END_VAR
VAR
  LastValue : INT ;
  Change : BOOL ;
  DirectionPlus : BOOL ;
  DirectionMinus : BOOL ;
  TimeStop : TIME  := T#500MS;
  Stop : BOOL ;
  StartTimer : BOOL ;
  delay : FB 185;
END_VAR
BEGIN
// body was compiled from another editor; compiled code not shown
END_FUNCTION_BLOCK

FUNCTION_BLOCK "Safety_Speed"	// FB 73
AUTHOR : Koenig
VERSION : 0.1
VAR_INPUT
  ActPosition : INT ;
END_VAR
VAR
  LastPositon : INT ;
  Differnce : INT ;
  SpeedSecond : INT ;
  Speed : INT ;
  NoChange : BOOL ;
  error : BOOL ;
  TimeStop : TIME  := T#500MS;
  SpeedNull : BOOL ;
  Speed_1 : INT ;
  Speed_2 : INT ;
  Speed_3 : INT ;
  Calc : INT ;
  Result : INT ;
  T_Stop : FB 185;
END_VAR
BEGIN
// body was compiled from another editor; compiled code not shown
END_FUNCTION_BLOCK

FUNCTION_BLOCK "Safety_SpeedCheck"	// FB 74
TITLE = Check safe speed speed
AUTHOR : Koenig
VERSION : 0.1
VAR_INPUT
  Reset : BOOL ;	//reset errors
  ReleaseFast : BOOL ;	//release fast speed
  CN_Stop : BOOL ;	//crane is not moving
  ActualSpeed : INT ;	//actual pseed in mm/s
  MaxSafeSpeed : INT ;	//max. safe speed in mm/s
  MaxSpeed : INT ;	//max. speed in mm/s
END_VAR
VAR_OUTPUT
  Error_SafeSpeed : BOOL ;
  Error_MaxSPeed : BOOL ;
END_VAR
VAR
  on : BOOL ;
  timeSafeSpeed : TIME  := T#4S;
  safeSpeed : BOOL ;
  nowCheck : BOOL ;
  DelayCheck : FB 185;
  err_SafeSpeed : BOOL ;
  err_Speed : BOOL ;
  err_OV : BOOL ;
  speed : INT ;
END_VAR
BEGIN
// body was compiled from another editor; compiled code not shown
END_FUNCTION_BLOCK

FUNCTION_BLOCK "Wago_Bridge"	// FB 80
TITLE = Check Hardware RBG Bridge
AUTHOR : Koenig
VERSION : 0.1
VAR_INPUT
  Reset : BOOL ;
END_VAR
VAR_OUTPUT
  HardwareOK : BOOL ;
END_VAR
VAR
  ON : BOOL ;
END_VAR
BEGIN
// body was compiled from another editor; compiled code not shown
END_FUNCTION_BLOCK

FUNCTION_BLOCK "F_Input_MAP"	// FB 91
TITLE = MAP safety input IOs (zones)
AUTHOR : Koenig
VERSION : 0.1
VAR
  ON : BOOL ;
  OFF : BOOL ;
  gblStopOK : BOOL ;
END_VAR
BEGIN
// body was compiled from another editor; compiled code not shown
END_FUNCTION_BLOCK

FUNCTION_BLOCK "ESTOP"	// FB 92
TITLE = ESTOP
AUTHOR : Koenig
VERSION : 0.1
VAR_INPUT
  Reset : BOOL ;
  Automatik : BOOL ;
END_VAR
VAR_OUTPUT
  ESTOP : BOOL ;
  ESTOP_DELAY : BOOL ;
END_VAR
VAR
  ON : BOOL ;
  Signal : BOOL ;
  M_ESTOP : BOOL ;
  Output : BOOL ;
  Q_Out_Delay : BOOL ;
  DelayEstop : FB 185;
END_VAR
BEGIN
// body was compiled from another editor; compiled code not shown
END_FUNCTION_BLOCK

FUNCTION_BLOCK "GetPos"	// FB 93
TITLE = Get position carier
AUTHOR : Koenig
VERSION : 0.1
VAR_INPUT
  AxisPos : INT ;
END_VAR
VAR_OUTPUT
  PosNo : INT ;
END_VAR
VAR
  iPos : INT ;
END_VAR
BEGIN
// body was compiled from another editor; compiled code not shown
END_FUNCTION_BLOCK

// FB 101: know-how protected block, not included

// FB 126: know-how protected block, not included

// FB 127: know-how protected block, not included

// FB 185: know-how protected block, not included

// FB 186: know-how protected block, not included

// FB 215: know-how protected block, not included

// FB 219: know-how protected block, not included

// FB 225: know-how protected block, not included

// FB 226: know-how protected block, not included

// FB 272: know-how protected block, not included

// FB 273: know-how protected block, not included

// FB 274: know-how protected block, not included

// FB 275: know-how protected block, not included

// FB 276: know-how protected block, not included

// FB 277: know-how protected block, not included

// FB 278: know-how protected block, not included

// FB 279: know-how protected block, not included

// FB 280: know-how protected block, not included

// FB 281: know-how protected block, not included

// FB 282: know-how protected block, not included

// FB 283: know-how protected block, not included

// FB 284: know-how protected block, not included

// FB 285: know-how protected block, not included

// FC 1: know-how protected block, not included

FUNCTION "Init" : VOID	// FC 2
TITLE = Program/PLC Init
VERSION : 0.1
BEGIN
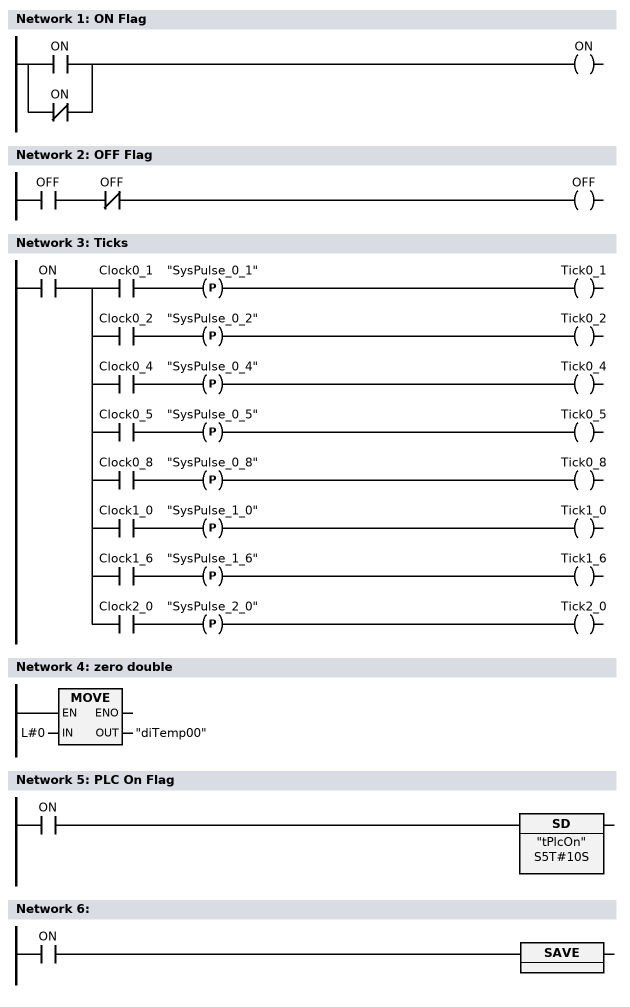
NETWORK
TITLE = ON Flag
      O     "ON";
      ON    "ON";
      =     "ON";
NETWORK
TITLE = OFF Flag
      A     "OFF";
      AN    "OFF";
      =     "OFF";
NETWORK
TITLE = Ticks
      A     "ON";
      =     L 0.0;
      A     L 0.0;
      A     "Clock0_1";
      FP    "SysPulse_0_1";
      =     "Tick0_1";
      A     L 0.0;
      A     "Clock0_2";
      FP    "SysPulse_0_2";
      =     "Tick0_2";
      A     L 0.0;
      A     "Clock0_4";
      FP    "SysPulse_0_4";
      =     "Tick0_4";
      A     L 0.0;
      A     "Clock0_5";
      FP    "SysPulse_0_5";
      =     "Tick0_5";
      A     L 0.0;
      A     "Clock0_8";
      FP    "SysPulse_0_8";
      =     "Tick0_8";
      A     L 0.0;
      A     "Clock1_0";
      FP    "SysPulse_1_0";
      =     "Tick1_0";
      A     L 0.0;
      A     "Clock1_6";
      FP    "SysPulse_1_6";
      =     "Tick1_6";
      A     L 0.0;
      A     "Clock2_0";
      FP    "SysPulse_2_0";
      =     "Tick2_0";
NETWORK
TITLE = zero double
      L     L#0;
      T     "diTemp00";
      NOP   0;
NETWORK
TITLE = PLC On Flag
      A     "ON";
      L     S5T#10S;
      SD    "tPlcOn";
NETWORK
TITLE =
      A     "ON";
      SAVE;
END_FUNCTION

// FC 5: know-how protected block, not included

// FC 6: know-how protected block, not included

// FC 8: know-how protected block, not included

FUNCTION "OpHours" : VOID	// FC 9
VERSION : 0.1
VAR_INPUT
  IN_xMoving : BOOL ;
  IN_xTick_1sec : BOOL ;
  IN_xResetServHours : BOOL ;
  IN_diServHoursPrest : DINT ;
END_VAR
VAR_IN_OUT
  INOUT_iWorkSec : INT ;
  INOUT_iServSec : INT ;
  INOUT_diWorkHours : DINT ;
  INOUT_diServHours : DINT ;
END_VAR
BEGIN
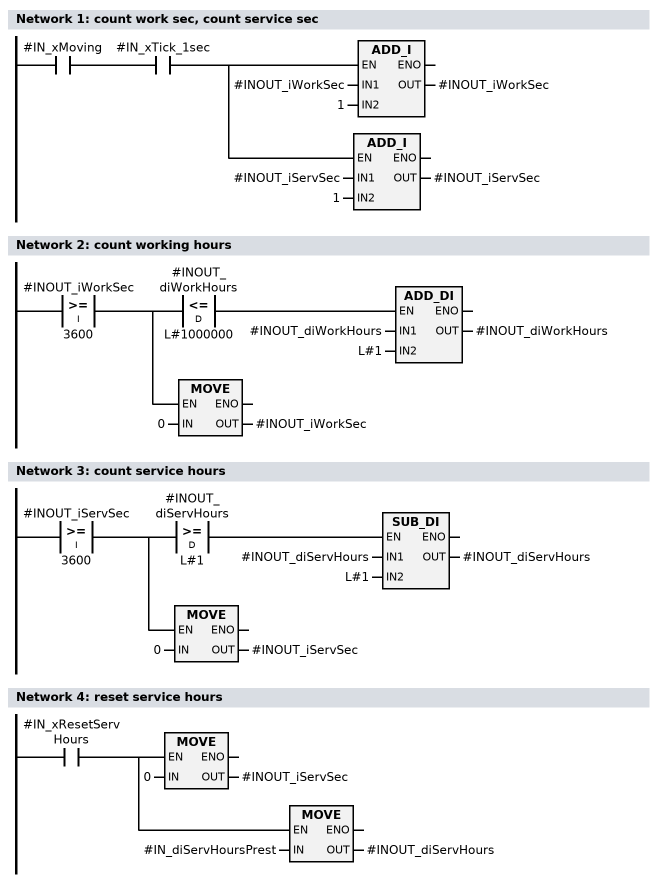
NETWORK
TITLE = count work sec, count service sec
      A     #IN_xMoving;
      A     #IN_xTick_1sec;
      =     L 0.0;
      A     L 0.0;
      JNB   _001;
      L     #INOUT_iWorkSec;
      L     1;
      +I;
      T     #INOUT_iWorkSec;
_001: NOP   0;
      A     L 0.0;
      JNB   _002;
      L     #INOUT_iServSec;
      L     1;
      +I;
      T     #INOUT_iServSec;
_002: NOP   0;
NETWORK
TITLE = count working hours
      L     #INOUT_iWorkSec;
      L     3600;
      >=I;
      =     L 0.0;
      A     L 0.0;
      A(;
      L     #INOUT_diWorkHours;
      L     L#1000000;
      <=D;
      );
      JNB   _003;
      L     #INOUT_diWorkHours;
      L     L#1;
      +D;
      T     #INOUT_diWorkHours;
_003: NOP   0;
      A     L 0.0;
      JNB   _004;
      L     0;
      T     #INOUT_iWorkSec;
_004: NOP   0;
NETWORK
TITLE = count service hours
      L     #INOUT_iServSec;
      L     3600;
      >=I;
      =     L 0.0;
      A     L 0.0;
      A(;
      L     #INOUT_diServHours;
      L     L#1;
      >=D;
      );
      JNB   _005;
      L     #INOUT_diServHours;
      L     L#1;
      -D;
      T     #INOUT_diServHours;
_005: NOP   0;
      A     L 0.0;
      JNB   _006;
      L     0;
      T     #INOUT_iServSec;
_006: NOP   0;
NETWORK
TITLE = reset service hours
      A     #IN_xResetServHours;
      =     L 0.0;
      A     L 0.0;
      JNB   _007;
      L     0;
      T     #INOUT_iServSec;
_007: NOP   0;
      A     L 0.0;
      JNB   _008;
      L     #IN_diServHoursPrest;
      T     #INOUT_diServHours;
_008: NOP   0;
END_FUNCTION

// FC 10: know-how protected block, not included

FUNCTION "AbsEncoder" : VOID	// FC 11
TITLE = AbsEncoder
//calculate position value depend from encoder resolution
VERSION : 0.1
VAR_INPUT
  IN_DW_ProcessData : DWORD ;
  IN_DINT_Turn100 : DINT ;
  IN_DINT_PresetVal : DINT ;
  IN_Resolution_4096 : BOOL ;
  IN_Resolution_8192 : BOOL ;
  IN_BOOL_Preset : BOOL ;
END_VAR
VAR_OUTPUT
  OUT_DINT_EncMm : DINT ;
  OUT_DW_ProcessData : DWORD ;
END_VAR
VAR_TEMP
  TEMP_DINT_WayByFullTurns : DINT ;
  TEMP_DINT_WayByActTurn : DINT ;
  TEMP_DINT_Resolution : DINT ;
  TEMP_DW_01 : DWORD ;
  TEMP_DW_00 : DWORD ;
  TEMP_DW_Mask1 : DWORD ;
  TEMP_W_Mask2 : WORD ;
  TEMP_DW_Mask3 : DWORD ;
  TEMP_DINT_00 : DINT ;
  TEMP_DINT_PresetTurns : DINT ;
  TEMP_DINT_PresetVal100 : DINT ;
  TEMP_DINT_PresetAngle : DINT ;
  ON : BOOL ;
  TEMP_BOOL_RetValFault : BOOL ;
END_VAR
BEGIN
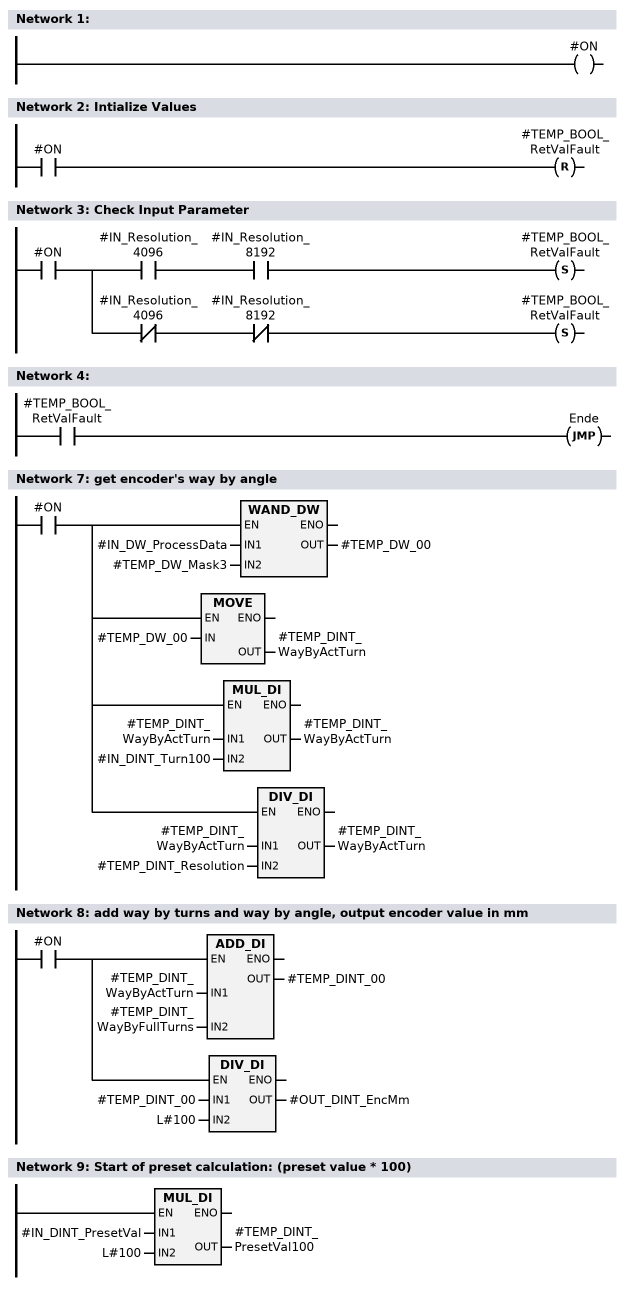
NETWORK
TITLE =
      SET;
      =     #ON;
NETWORK
TITLE = Intialize Values
      A     #ON;
      R     #TEMP_BOOL_RetValFault;
NETWORK
TITLE = Check Input Parameter
      A     #ON;
      =     L 47.0;
      A     L 47.0;
      A     #IN_Resolution_4096;
      A     #IN_Resolution_8192;
      S     #TEMP_BOOL_RetValFault;
      A     L 47.0;
      AN    #IN_Resolution_4096;
      AN    #IN_Resolution_8192;
      S     #TEMP_BOOL_RetValFault;
NETWORK
TITLE =
      A     #TEMP_BOOL_RetValFault;
      JC    Ende;
NETWORK
TITLE =
      A     #ON;
      =     L 47.0;
      A     L 47.0;
      A     #IN_Resolution_4096;
      =     L 47.1;
      A(;
      A(;
      A     L 47.1;
      JNB   _001;
      L     DW#16#1FFF000;
      T     #TEMP_DW_Mask1;
      SET;
      SAVE;
      CLR;
_001: A     BR;
      );
      JNB   _002;
      L     W#16#C;
      T     #TEMP_W_Mask2;
      SET;
      SAVE;
      CLR;
_002: A     BR;
      );
      JNB   _003;
      L     DW#16#FFF;
      T     #TEMP_DW_Mask3;
_003: NOP   0;
      A     L 47.1;
      JNB   _004;
      L     L#4096;
      T     #TEMP_DINT_Resolution;
_004: NOP   0;
      A     L 47.0;
      A     #IN_Resolution_8192;
      =     L 47.1;
      A(;
      A(;
      A     L 47.1;
      JNB   _005;
      L     DW#16#1FFE000;
      T     #TEMP_DW_Mask1;
      SET;
      SAVE;
      CLR;
_005: A     BR;
      );
      JNB   _006;
      L     W#16#D;
      T     #TEMP_W_Mask2;
      SET;
      SAVE;
      CLR;
_006: A     BR;
      );
      JNB   _007;
      L     DW#16#1FFF;
      T     #TEMP_DW_Mask3;
_007: NOP   0;
      A     L 47.1;
      JNB   _008;
      L     L#8192;
      T     #TEMP_DINT_Resolution;
_008: NOP   0;
NETWORK
TITLE = Start of actual mm-calculation: get encoder's way by full turns
      A     #ON;
      =     L 47.0;
      A     L 47.0;
      JNB   _009;
      L     #IN_DW_ProcessData;
      L     #TEMP_DW_Mask1;
      AD;
      T     #TEMP_DW_00;
_009: NOP   0;
      A     L 47.0;
      JNB   _00a;
      L     #TEMP_W_Mask2;
      L     #TEMP_DW_00;
      SRD;
      T     #TEMP_DW_00;
_00a: NOP   0;
      A     L 47.0;
      JNB   _00b;
      L     #TEMP_DW_00;
      T     #TEMP_DINT_WayByFullTurns;
_00b: NOP   0;
      A     L 47.0;
      JNB   _00c;
      L     #TEMP_DINT_WayByFullTurns;
      L     #IN_DINT_Turn100;
      *D;
      T     #TEMP_DINT_WayByFullTurns;
_00c: NOP   0;
NETWORK
TITLE = get encoder's way by angle
      A     #ON;
      =     L 47.0;
      A     L 47.0;
      JNB   _00d;
      L     #IN_DW_ProcessData;
      L     #TEMP_DW_Mask3;
      AD;
      T     #TEMP_DW_00;
_00d: NOP   0;
      A     L 47.0;
      JNB   _00e;
      L     #TEMP_DW_00;
      T     #TEMP_DINT_WayByActTurn;
_00e: NOP   0;
      A     L 47.0;
      JNB   _00f;
      L     #TEMP_DINT_WayByActTurn;
      L     #IN_DINT_Turn100;
      *D;
      T     #TEMP_DINT_WayByActTurn;
_00f: NOP   0;
      A     L 47.0;
      JNB   _010;
      L     #TEMP_DINT_WayByActTurn;
      L     #TEMP_DINT_Resolution;
      /D;
      T     #TEMP_DINT_WayByActTurn;
_010: NOP   0;
NETWORK
TITLE = add way by turns and way by angle, output encoder value in mm
      A     #ON;
      =     L 47.0;
      A     L 47.0;
      JNB   _011;
      L     #TEMP_DINT_WayByActTurn;
      L     #TEMP_DINT_WayByFullTurns;
      +D;
      T     #TEMP_DINT_00;
_011: NOP   0;
      A     L 47.0;
      JNB   _012;
      L     #TEMP_DINT_00;
      L     L#100;
      /D;
      T     #OUT_DINT_EncMm;
_012: NOP   0;
NETWORK
TITLE = Start of preset calculation: (preset value * 100)
      L     #IN_DINT_PresetVal;
      L     L#100;
      *D;
      T     #TEMP_DINT_PresetVal100;
      NOP   0;
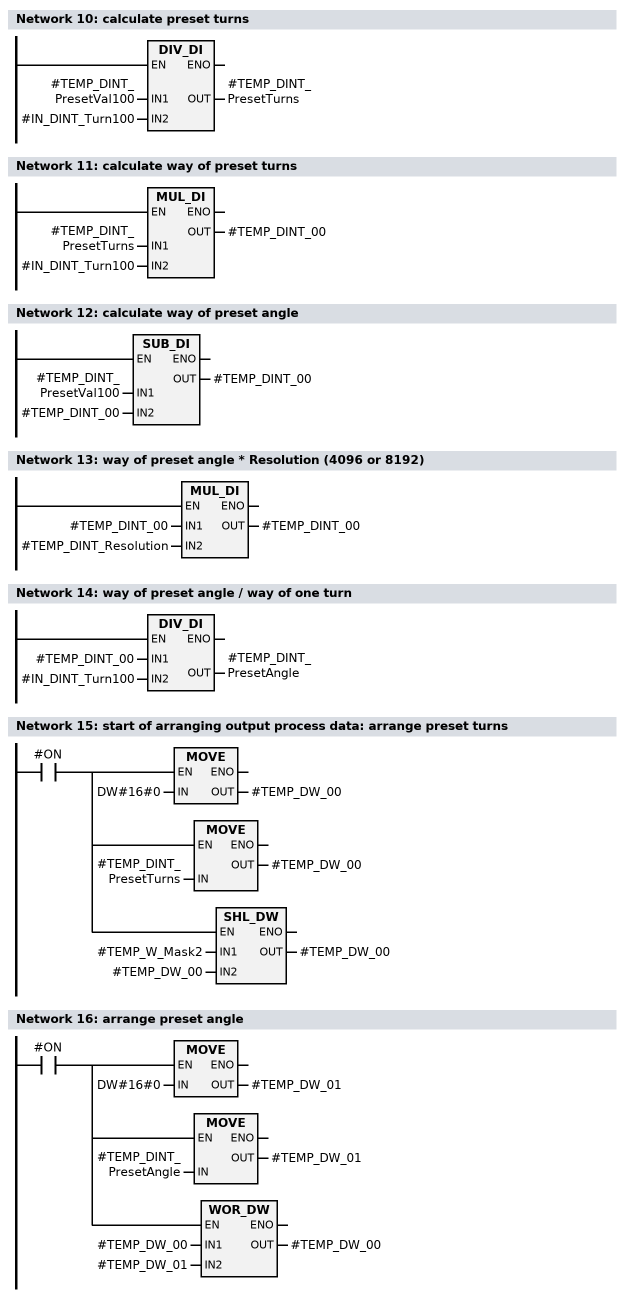
NETWORK
TITLE = calculate preset turns
      L     #TEMP_DINT_PresetVal100;
      L     #IN_DINT_Turn100;
      /D;
      T     #TEMP_DINT_PresetTurns;
      NOP   0;
NETWORK
TITLE = calculate way of preset turns
      L     #TEMP_DINT_PresetTurns;
      L     #IN_DINT_Turn100;
      *D;
      T     #TEMP_DINT_00;
      NOP   0;
NETWORK
TITLE = calculate way of preset angle 
      L     #TEMP_DINT_PresetVal100;
      L     #TEMP_DINT_00;
      -D;
      T     #TEMP_DINT_00;
      NOP   0;
NETWORK
TITLE = way of preset angle * Resolution (4096 or 8192)
      L     #TEMP_DINT_00;
      L     #TEMP_DINT_Resolution;
      *D;
      T     #TEMP_DINT_00;
      NOP   0;
NETWORK
TITLE = way of preset angle / way of one turn
      L     #TEMP_DINT_00;
      L     #IN_DINT_Turn100;
      /D;
      T     #TEMP_DINT_PresetAngle;
      NOP   0;
NETWORK
TITLE = start of arranging output process data: arrange preset turns
      A     #ON;
      =     L 47.0;
      A     L 47.0;
      JNB   _013;
      L     DW#16#0;
      T     #TEMP_DW_00;
_013: NOP   0;
      A     L 47.0;
      JNB   _014;
      L     #TEMP_DINT_PresetTurns;
      T     #TEMP_DW_00;
_014: NOP   0;
      A     L 47.0;
      JNB   _015;
      L     #TEMP_W_Mask2;
      L     #TEMP_DW_00;
      SLD;
      T     #TEMP_DW_00;
_015: NOP   0;
NETWORK
TITLE = arrange preset angle
      A     #ON;
      =     L 47.0;
      A     L 47.0;
      JNB   _016;
      L     DW#16#0;
      T     #TEMP_DW_01;
_016: NOP   0;
      A     L 47.0;
      JNB   _017;
      L     #TEMP_DINT_PresetAngle;
      T     #TEMP_DW_01;
_017: NOP   0;
      A     L 47.0;
      JNB   _018;
      L     #TEMP_DW_00;
      L     #TEMP_DW_01;
      OD;
      T     #TEMP_DW_00;
_018: NOP   0;
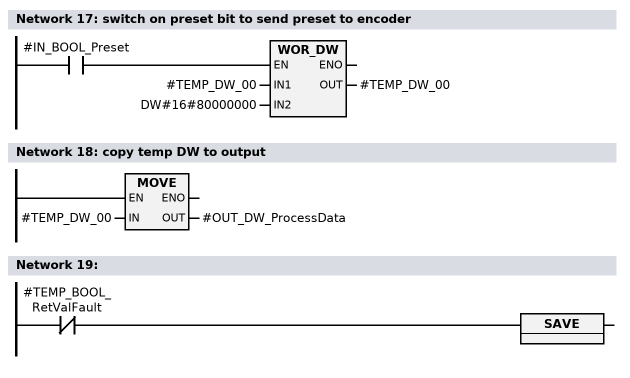
NETWORK
TITLE = switch on preset bit to send preset to encoder
      A     #IN_BOOL_Preset;
      JNB   _019;
      L     #TEMP_DW_00;
      L     DW#16#80000000;
      OD;
      T     #TEMP_DW_00;
_019: NOP   0;
NETWORK
TITLE = copy temp DW to output 
      L     #TEMP_DW_00;
      T     #OUT_DW_ProcessData;
      NOP   0;
NETWORK
TITLE =
Ende: AN    #TEMP_BOOL_RetValFault;
      SAVE;
END_FUNCTION

// FC 15: know-how protected block, not included

FUNCTION "Inputs" : VOID	// FC 30
TITLE = Inputs
VERSION : 0.1
VAR_TEMP
  tmp_Retval : INT ;
  tmp_d : INT ;
  tmp_u : DINT ;
  value : INT ;
  d_value : DINT ;
END_VAR
BEGIN
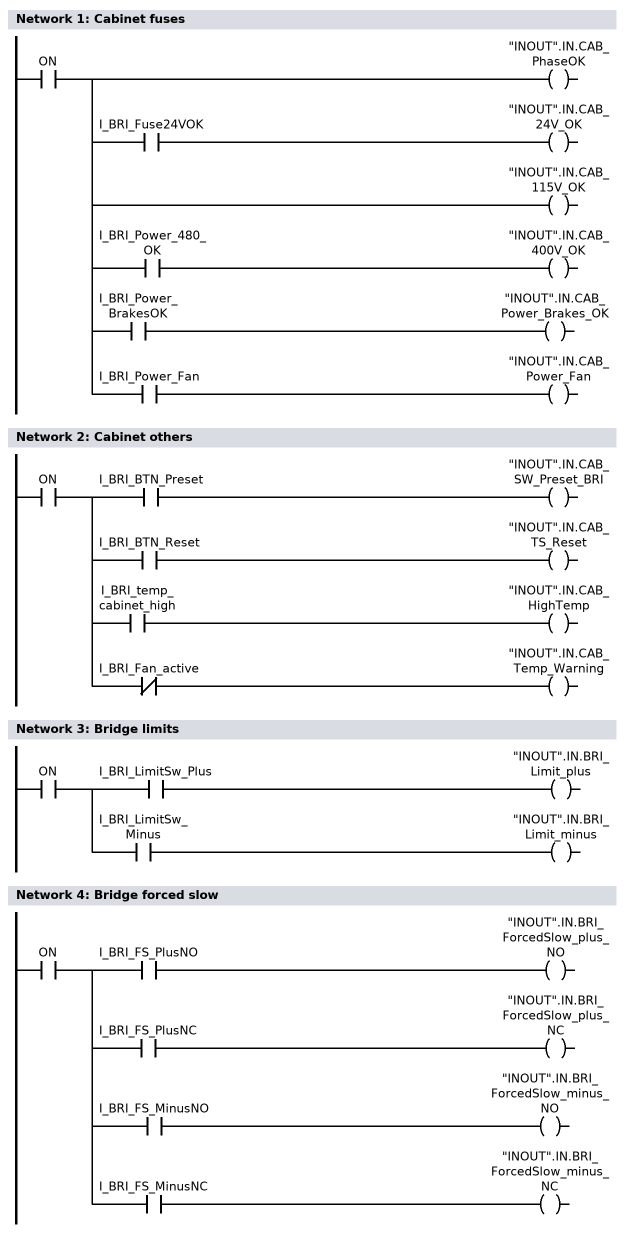
NETWORK
TITLE = Cabinet fuses
      A     "ON";
      =     L 14.0;
      A     L 14.0;
      BLD   102;
      =     "INOUT".IN.CAB_PhaseOK;
      A     L 14.0;
      A     "I_BRI_Fuse24VOK";
      =     "INOUT".IN.CAB_24V_OK;
      A     L 14.0;
      BLD   102;
      =     "INOUT".IN.CAB_115V_OK;
      A     L 14.0;
      A     "I_BRI_Power_480_OK";
      =     "INOUT".IN.CAB_400V_OK;
      A     L 14.0;
      A     "I_BRI_Power_BrakesOK";
      =     "INOUT".IN.CAB_Power_Brakes_OK;
      A     L 14.0;
      A     "I_BRI_Power_Fan";
      =     "INOUT".IN.CAB_Power_Fan;
NETWORK
TITLE = Cabinet others
      A     "ON";
      =     L 14.0;
      A     L 14.0;
      A     "I_BRI_BTN_Preset";
      =     "INOUT".IN.CAB_SW_Preset_BRI;
      A     L 14.0;
      A     "I_BRI_BTN_Reset";
      =     "INOUT".IN.CAB_TS_Reset;
      A     L 14.0;
      A     "I_BRI_temp_cabinet_high";
      =     "INOUT".IN.CAB_HighTemp;
      A     L 14.0;
      AN    "I_BRI_Fan_active";
      =     "INOUT".IN.CAB_Temp_Warning;
NETWORK
TITLE = Bridge limits
      A     "ON";
      =     L 14.0;
      A     L 14.0;
      A     "I_BRI_LimitSw_Plus";
      =     "INOUT".IN.BRI_Limit_plus;
      A     L 14.0;
      A     "I_BRI_LimitSw_Minus";
      =     "INOUT".IN.BRI_Limit_minus;
NETWORK
TITLE = Bridge forced slow
      A     "ON";
      =     L 14.0;
      A     L 14.0;
      A     "I_BRI_FS_PlusNO";
      =     "INOUT".IN.BRI_ForcedSlow_plus_NO;
      A     L 14.0;
      A     "I_BRI_FS_PlusNC";
      =     "INOUT".IN.BRI_ForcedSlow_plus_NC;
      A     L 14.0;
      A     "I_BRI_FS_MinusNO";
      =     "INOUT".IN.BRI_ForcedSlow_minus_NO;
      A     L 14.0;
      A     "I_BRI_FS_MinusNC";
      =     "INOUT".IN.BRI_ForcedSlow_minus_NC;
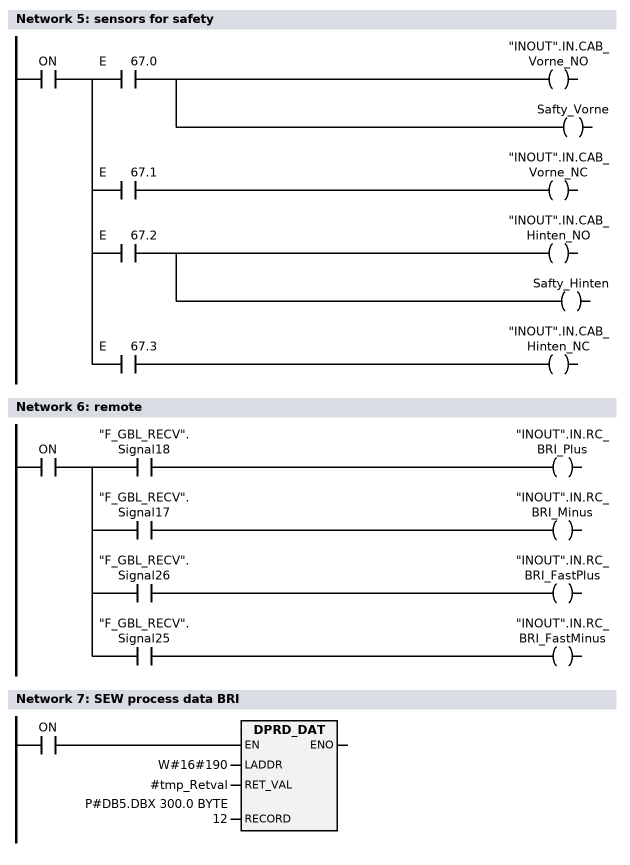
NETWORK
TITLE = sensors for safety
      A     "ON";
      =     L 14.0;
      A     L 14.0;
      A     "E      67.0";
      =     "INOUT".IN.CAB_Vorne_NO;
      =     "Safty_Vorne";
      A     L 14.0;
      A     "E      67.1";
      =     "INOUT".IN.CAB_Vorne_NC;
      A     L 14.0;
      A     "E      67.2";
      =     "INOUT".IN.CAB_Hinten_NO;
      =     "Safty_Hinten";
      A     L 14.0;
      A     "E      67.3";
      =     "INOUT".IN.CAB_Hinten_NC;
NETWORK
TITLE = remote
      A     "ON";
      =     L 14.0;
      A     L 14.0;
      A     "F_GBL_RECV".Signal18;
      =     "INOUT".IN.RC_BRI_Plus;
      A     L 14.0;
      A     "F_GBL_RECV".Signal17;
      =     "INOUT".IN.RC_BRI_Minus;
      A     L 14.0;
      A     "F_GBL_RECV".Signal26;
      =     "INOUT".IN.RC_BRI_FastPlus;
      A     L 14.0;
      A     "F_GBL_RECV".Signal25;
      =     "INOUT".IN.RC_BRI_FastMinus;
NETWORK
TITLE = SEW process data BRI
//PEW400 = 190h
      A     "ON";
      JNB   _001;
      CALL  "DPRD_DAT" (
           LADDR                    := W#16#190,
           RET_VAL                  := #tmp_Retval,
           RECORD                   := P#DB5.DBX 300.0 BYTE 12);
_001: NOP   0;
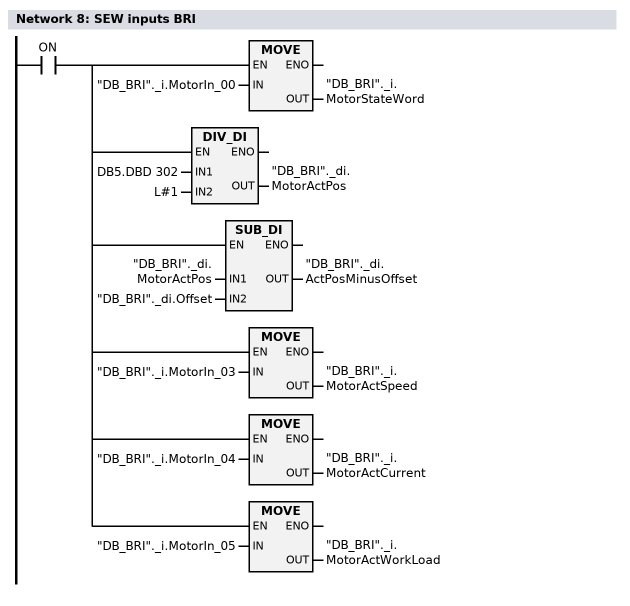
NETWORK
TITLE = SEW inputs BRI
      A     "ON";
      =     L 14.0;
      A     L 14.0;
      JNB   _002;
      L     "DB_BRI"._i.MotorIn_00;
      T     "DB_BRI"._i.MotorStateWord;
_002: NOP   0;
      A     L 14.0;
      JNB   _003;
      L     DB5.DBD 302;
      L     L#1;
      /D;
      T     "DB_BRI"._di.MotorActPos;
_003: NOP   0;
      A     L 14.0;
      JNB   _004;
      L     "DB_BRI"._di.MotorActPos;
      L     "DB_BRI"._di.Offset;
      -D;
      T     "DB_BRI"._di.ActPosMinusOffset;
_004: NOP   0;
      A     L 14.0;
      JNB   _005;
      L     "DB_BRI"._i.MotorIn_03;
      T     "DB_BRI"._i.MotorActSpeed;
_005: NOP   0;
      A     L 14.0;
      JNB   _006;
      L     "DB_BRI"._i.MotorIn_04;
      T     "DB_BRI"._i.MotorActCurrent;
_006: NOP   0;
      A     L 14.0;
      JNB   _007;
      L     "DB_BRI"._i.MotorIn_05;
      T     "DB_BRI"._i.MotorActWorkLoad;
_007: NOP   0;
END_FUNCTION

FUNCTION "Outputs" : VOID	// FC 31
TITLE = Outputs
VERSION : 0.1
VAR_TEMP
  tmp_Retval : INT ;
END_VAR
BEGIN
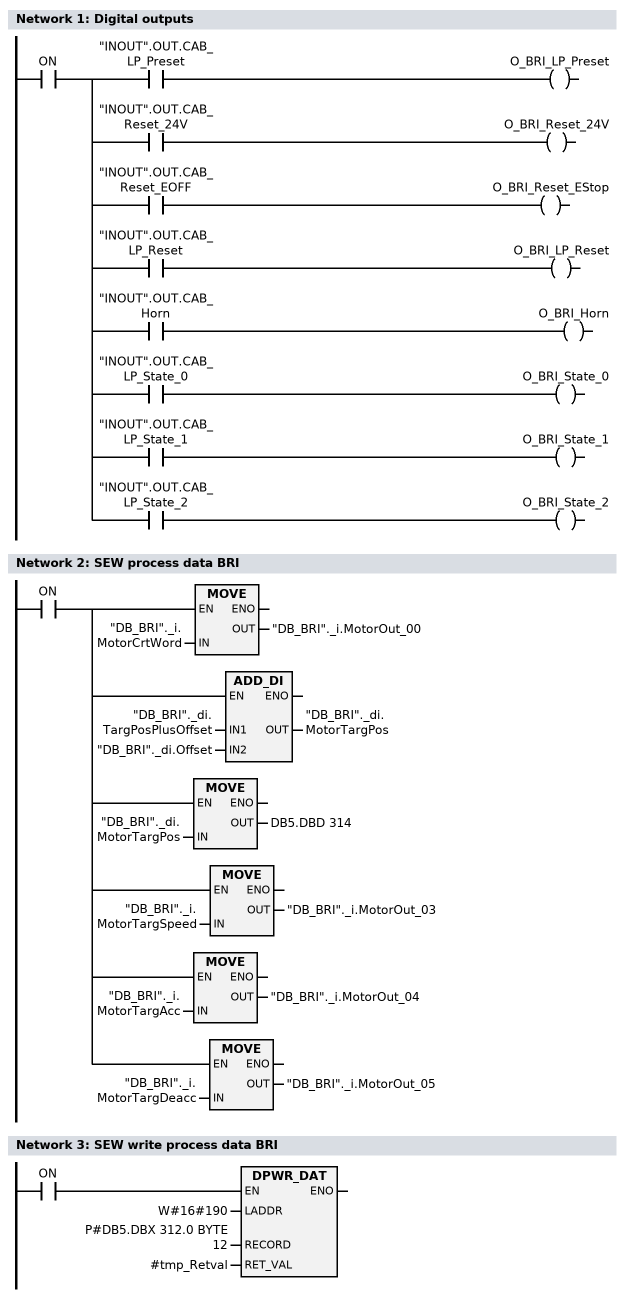
NETWORK
TITLE = Digital outputs
      A     "ON";
      =     L 2.0;
      A     L 2.0;
      A     "INOUT".OUT.CAB_LP_Preset;
      =     "O_BRI_LP_Preset";
      A     L 2.0;
      A     "INOUT".OUT.CAB_Reset_24V;
      =     "O_BRI_Reset_24V";
      A     L 2.0;
      A     "INOUT".OUT.CAB_Reset_EOFF;
      =     "O_BRI_Reset_EStop";
      A     L 2.0;
      A     "INOUT".OUT.CAB_LP_Reset;
      =     "O_BRI_LP_Reset";
      A     L 2.0;
      A     "INOUT".OUT.CAB_Horn;
      =     "O_BRI_Horn";
      A     L 2.0;
      A     "INOUT".OUT.CAB_LP_State_0;
      =     "O_BRI_State_0";
      A     L 2.0;
      A     "INOUT".OUT.CAB_LP_State_1;
      =     "O_BRI_State_1";
      A     L 2.0;
      A     "INOUT".OUT.CAB_LP_State_2;
      =     "O_BRI_State_2";
NETWORK
TITLE = SEW process data BRI
      A     "ON";
      =     L 2.0;
      A     L 2.0;
      JNB   _001;
      L     "DB_BRI"._i.MotorCrtWord;
      T     "DB_BRI"._i.MotorOut_00;
_001: NOP   0;
      A     L 2.0;
      JNB   _002;
      L     "DB_BRI"._di.TargPosPlusOffset;
      L     "DB_BRI"._di.Offset;
      +D;
      T     "DB_BRI"._di.MotorTargPos;
_002: NOP   0;
      A     L 2.0;
      JNB   _003;
      L     "DB_BRI"._di.MotorTargPos;
      T     DB5.DBD 314;
_003: NOP   0;
      A     L 2.0;
      JNB   _004;
      L     "DB_BRI"._i.MotorTargSpeed;
      T     "DB_BRI"._i.MotorOut_03;
_004: NOP   0;
      A     L 2.0;
      JNB   _005;
      L     "DB_BRI"._i.MotorTargAcc;
      T     "DB_BRI"._i.MotorOut_04;
_005: NOP   0;
      A     L 2.0;
      JNB   _006;
      L     "DB_BRI"._i.MotorTargDeacc;
      T     "DB_BRI"._i.MotorOut_05;
_006: NOP   0;
NETWORK
TITLE = SEW write process data BRI
//PEW400 = 190h
      A     "ON";
      JNB   _007;
      CALL  "DPWR_DAT" (
           LADDR                    := W#16#190,
           RECORD                   := P#DB5.DBX 312.0 BYTE 12,
           RET_VAL                  := #tmp_Retval);
_007: NOP   0;
END_FUNCTION

FUNCTION "Errors" : VOID	// FC 40
TITLE = Errors
VERSION : 0.1
BEGIN
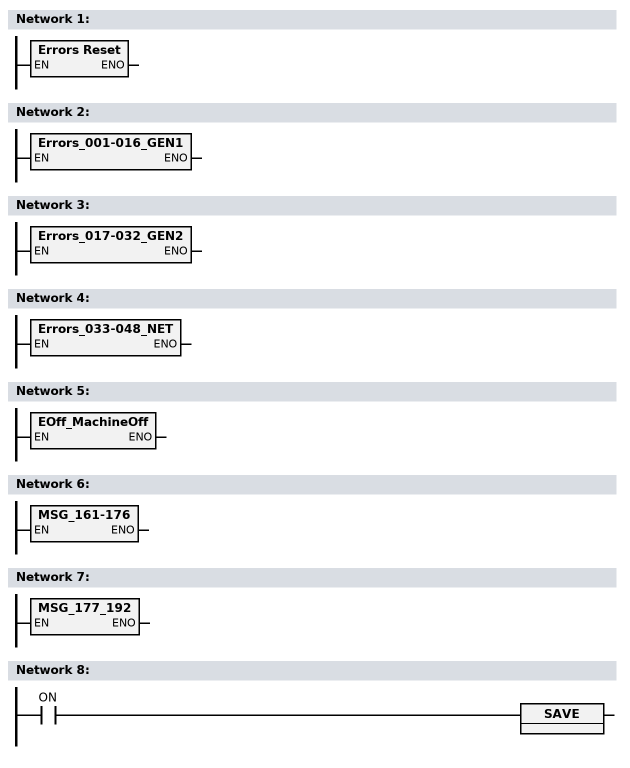
NETWORK
TITLE =
      CALL  "Errors Reset";
      NOP   0;
NETWORK
TITLE =
      CALL  "Errors_001-016_GEN1";
      NOP   0;
NETWORK
TITLE =
      CALL  "Errors_017-032_GEN2";
      NOP   0;
NETWORK
TITLE =
      CALL  "Errors_033-048_NET";
      NOP   0;
NETWORK
TITLE =
      CALL  "EOff_MachineOff";
      NOP   0;
NETWORK
TITLE =
      CALL  "MSG_161-176";
      NOP   0;
NETWORK
TITLE =
      CALL  "MSG_177_192";
      NOP   0;
NETWORK
TITLE =
      A     "ON";
      SAVE;
END_FUNCTION

FUNCTION "Errors Reset" : VOID	// FC 41
TITLE = Errors Reset
VERSION : 0.1
VAR_TEMP
  tmp_RetVal : INT ;
END_VAR
BEGIN
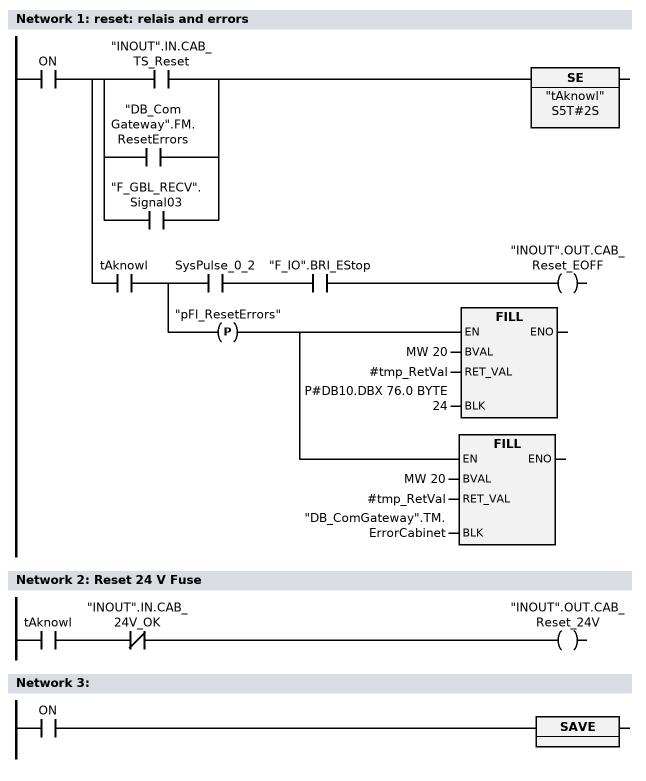
NETWORK
TITLE = reset: relais and errors
      A     "ON";
      =     L 2.0;
      A     L 2.0;
      A(;
      O     "INOUT".IN.CAB_TS_Reset;
      O     "DB_ComGateway".FM.ResetErrors;
      O     "F_GBL_RECV".Signal03;
      );
      L     S5T#2S;
      SE    "tAknowl";
      A     L 2.0;
      A     "tAknowl";
      =     L 2.1;
      A     L 2.1;
      A     "SysPulse_0_2";
      A     "F_IO".BRI_EStop;
      =     "INOUT".OUT.CAB_Reset_EOFF;
      A     L 2.1;
      FP    "pFl_ResetErrors";
      =     L 2.2;
      A     L 2.2;
      JNB   _001;
      CALL  "FILL" (
           BVAL                     := MW 20,
           RET_VAL                  := #tmp_RetVal,
           BLK                      := P#DB10.DBX 76.0 BYTE 24);
_001: NOP   0;
      A     L 2.2;
      JNB   _002;
      CALL  "FILL" (
           BVAL                     := MW 20,
           RET_VAL                  := #tmp_RetVal,
           BLK                      := "DB_ComGateway".TM.ErrorCabinet);
_002: NOP   0;
NETWORK
TITLE = Reset 24 V Fuse
      A     "tAknowl";
      AN    "INOUT".IN.CAB_24V_OK;
      =     "INOUT".OUT.CAB_Reset_24V;
NETWORK
TITLE =
      A     "ON";
      SAVE;
END_FUNCTION

FUNCTION "Errors_001-016_GEN1" : VOID	// FC 42
TITLE = Errors GEN1
VERSION : 0.1
BEGIN
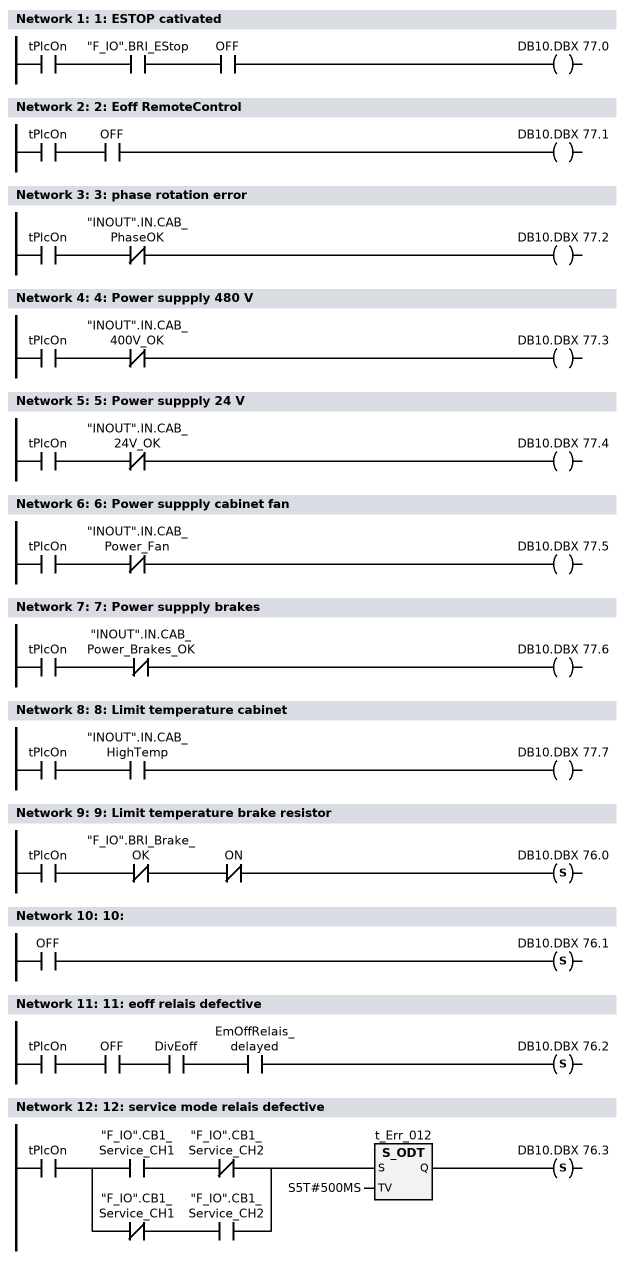
NETWORK
TITLE = 1: ESTOP cativated
      A     "tPlcOn";
      A     "F_IO".BRI_EStop;
      A     "OFF";
      =     DB10.DBX 77.0;
NETWORK
TITLE = 2: Eoff RemoteControl
      A     "tPlcOn";
      A     "OFF";
      =     DB10.DBX 77.1;
NETWORK
TITLE = 3: phase rotation error
      A     "tPlcOn";
      AN    "INOUT".IN.CAB_PhaseOK;
      =     DB10.DBX 77.2;
NETWORK
TITLE = 4: Power suppply 480 V
      A     "tPlcOn";
      AN    "INOUT".IN.CAB_400V_OK;
      =     DB10.DBX 77.3;
NETWORK
TITLE = 5: Power suppply 24 V
      A     "tPlcOn";
      AN    "INOUT".IN.CAB_24V_OK;
      =     DB10.DBX 77.4;
NETWORK
TITLE = 6: Power suppply cabinet fan
      A     "tPlcOn";
      AN    "INOUT".IN.CAB_Power_Fan;
      =     DB10.DBX 77.5;
NETWORK
TITLE = 7: Power suppply brakes
      A     "tPlcOn";
      AN    "INOUT".IN.CAB_Power_Brakes_OK;
      =     DB10.DBX 77.6;
NETWORK
TITLE = 8: Limit temperature cabinet
      A     "tPlcOn";
      A     "INOUT".IN.CAB_HighTemp;
      =     DB10.DBX 77.7;
NETWORK
TITLE = 9: Limit temperature brake resistor
      A     "tPlcOn";
      AN    "F_IO".BRI_Brake_OK;
      AN    "ON";
      S     DB10.DBX 76.0;
NETWORK
TITLE = 10:
      A     "OFF";
      S     DB10.DBX 76.1;
NETWORK
TITLE = 11: eoff relais defective
      A     "tPlcOn";
      A     "OFF";
      A     "DivEoff";
      A     "EmOffRelais_delayed";
      S     DB10.DBX 76.2;
NETWORK
TITLE = 12: service mode relais defective
      A     "tPlcOn";
      A(;
      A     "F_IO".CB1_Service_CH1;
      AN    "F_IO".CB1_Service_CH2;
      O;
      AN    "F_IO".CB1_Service_CH1;
      A     "F_IO".CB1_Service_CH2;
      );
      L     S5T#500MS;
      SD    "t_Err_012";
      NOP   0;
      NOP   0;
      NOP   0;
      A     "t_Err_012";
      S     DB10.DBX 76.3;
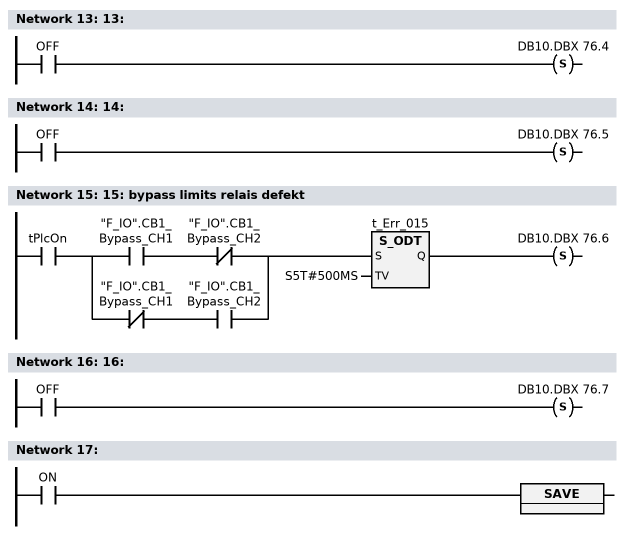
NETWORK
TITLE = 13:
      A     "OFF";
      S     DB10.DBX 76.4;
NETWORK
TITLE = 14:
      A     "OFF";
      S     DB10.DBX 76.5;
NETWORK
TITLE = 15: bypass limits relais defekt
      A     "tPlcOn";
      A(;
      A     "F_IO".CB1_Bypass_CH1;
      AN    "F_IO".CB1_Bypass_CH2;
      O;
      AN    "F_IO".CB1_Bypass_CH1;
      A     "F_IO".CB1_Bypass_CH2;
      );
      L     S5T#500MS;
      SD    "t_Err_015";
      NOP   0;
      NOP   0;
      NOP   0;
      A     "t_Err_015";
      S     DB10.DBX 76.6;
NETWORK
TITLE = 16:
      A     "OFF";
      S     DB10.DBX 76.7;
NETWORK
TITLE =
      A     "ON";
      SAVE;
END_FUNCTION

FUNCTION "Errors_017-032_GEN2" : VOID	// FC 43
TITLE = Errors GEN2
VERSION : 0.1
BEGIN
